(* CODESYS project mbc_Log4TC_tc3-4024_v0.2.1.library
   DefaultNamespace: log4tc
   DocFormat: reStructuredText
   Description: A library for logging in PLC code.
   Author: mbc engineering GmbH
   Title: log4TC
   Version: 0.2.1
   Company: mbc engineering GmbH
   Placeholder: log4TC

Project tree, tasks and I/O mapping:
  libraries: Base Interfaces, * (System); Tc2_Standard, * (Beckhoff Automation GmbH); Tc2_System, * (Beckhoff Automation GmbH); Tc2_Utilities, * (Beckhoff Automation GmbH); Tc3_Module, * (Beckhoff Automation GmbH); TcUnit, 1.0.0.0 (www.tcunit.org)
  API/
    Context/
      function F_LogContext [ST]
      function block FB_ScopedContext [ST]: Begin, ContextBuilder, End
      interface I_ContextBuilder: AddBool, AddByte, AddDInt, AddDWord, AddInt, AddLint, AddLReal, AddLWord, AddReal, AddSInt, AddString, AddUDInt, AddUInt, AddULint, AddUSInt, AddWord, Clear, Remove
    Full/
      function block FB_LoggerLAC [ST]: FB_init, LoggerContext
    Simple/
      Any/
        function F_LogA1 [ST]
        function F_LogA10 [ST]
        function F_LogA2 [ST]
        function F_LogA3 [ST]
        function F_LogA4 [ST]
        function F_LogA5 [ST]
        function F_LogA6 [ST]
        function F_LogA7 [ST]
        function F_LogA8 [ST]
        function F_LogA9 [ST]
        function F_LogLA1 [ST]
        function F_LogLA10 [ST]
        function F_LogLA10C [ST]
        function F_LogLA1C [ST]
        function F_LogLA2 [ST]
        function F_LogLA2C [ST]
        function F_LogLA3 [ST]
        function F_LogLA3C [ST]
        function F_LogLA4 [ST]
        function F_LogLA4C [ST]
        function F_LogLA5 [ST]
        function F_LogLA5C [ST]
        function F_LogLA6 [ST]
        function F_LogLA6C [ST]
        function F_LogLA7 [ST]
        function F_LogLA7C [ST]
        function F_LogLA8 [ST]
        function F_LogLA8C [ST]
        function F_LogLA9 [ST]
        function F_LogLA9C [ST]
      TArg/
        function F_LogL1 [ST]
        function F_LogL10 [ST]
        function F_LogL2 [ST]
        function F_LogL3 [ST]
        function F_LogL4 [ST]
        function F_LogL5 [ST]
        function F_LogL6 [ST]
        function F_LogL7 [ST]
        function F_LogL8 [ST]
        function F_LogL9 [ST]
      function F_Log [ST]
      function F_LogBuilder [ST]
      function F_LogC [ST]
      function F_LogL [ST]
      function F_LogLC [ST]
      interface I_LogBuilder: CreateLog, WithContextInt, WithIntArg, WithLogger, WithStringArg
    data type E_LogLevel
    program PRG_TaskLog [ST]: Call, Init, RtcTime, TaskContextBuilder, TaskLogger
  DUTs/
    data type E_CustomTypes
    data type E_Scope
    data type ST_Log4TcTaskInfo
    data type ST_ScopedContextStack
  GVLs/
    global variables Config
    global variables Const
    global variables Log4TcInfo
  ITFs/
    interface I_LogEntryAdder: AddToLogEntry
  POUs/
    Utils/
      function F_DINT_TO_UINT_MAX [ST]
      function block FB_LogBuffer [ST]: BufferFree, BufferPtr, BufferStartPtr, BufferUsed, Clear, DataAdded
      function block FB_RTC_Sync [ST]: Call, RtcTime
      function IncUDINT [ST]
    function F_InternalLog [ST]
    function F_LogA [ST]
    function F_LogTArg [ST]
    function block FB_ContextBuilder [ST]: _FindContext, _GetDataLen, _GetOffsetToData, _GetSize, _ReadName, _ReadType, AddBool, AddByte, AddDInt, AddDWord, AddInt, AddLInt, AddLReal, AddLWord, AddReal, AddSInt, AddString, AddUDInt, AddUInt, AddULInt, AddUSInt, AddWord, Clear, Remove, _BufferCount, _ContextCount, _GetContextOffset, _AddContext, _Copy, _RemoveContext, _ReplaceContext, _Reset, _WriteByte, _WriteInt, AddToLogEntry
    function block FB_Log4TcTask [ST]: _InitAndCheckTask, _ReadBuffer, Call, Init, TaskContext, WriteBuffer
    function block FB_LogEntry [ST]: _Copy, _Reset, _WriteByte, _WriteDInt, _WriteInt, _WriteLInt, _WriteString, _WriteUDInt, _WriteUInt, _WriteWString, AddAnyArg, AddBuffer, AddContext, AddTArg, End, Start
    program PRG_ScopedContextStack [ST]: TaskContextStack
  Test/
    function block FB_ContextBuilder_Test [ST]: AddInt_ShouldAddInt, AddInt_WithSameName_ShouldReplace, AddString_ShouldAddString, AddString_WithSameName_ShouldReAdd, AddString_WithSameName_ShouldReplace, RemoveInt_ShouldRemove, RemoveString_ShouldRemove
    program PRG_Test [ST]
  Version/
    global variables Global_Version
  program ApiTest [ST]
*)

// API/E_LogLevel
(*
:Description: Definition of available log levels. 

The log levels are ordered. ``eTrace`` has the lowest priority, ``eFatal`` has the
highest priority.

===============
Log Level Usage
===============

Is is recommended to build a guidline for consistent use of the log level. A example
could be the following:

:eFatal: The fatal level should be used for any error which will to malfunction of the most
	part of the program. Log message of this type must be handled immedialtely.
	
	Example: A Safety controller could not be initialised

:eError: The error level should be used when the program cannot continue to work properly.
	Normally this means that a operator/user has to be alerted and something has to
	be fixed.

	Example: Communication errors, something stops a process

:eWarn: The warn level should be used when some expected condition has happend, but the
	software can proceed in some way or the operation can be repeated later. Normaly
	the warn level should be read by the user/operator at some time, not necessarly 
	immediately.

	Example: Cannot connect to some external system (but will repeat to try)

:eInfo: The info level should track some of the import state changes in the programm. This
	information can be used by the user/operator on demand to track a problem.

	Example: A state of a state-machine has changed, a new recipe has been loaded

:eDebug: The info level should track of the some internals, normally only of importance to
	developers.

:eTrace: The trace level should be used to track some internal processing. This is rarely
	used, even by developers, mostly to track some difficult problem.

*)
{attribute 'qualified_only'}
{attribute 'strict'}
{attribute 'to_string'}
TYPE E_LogLevel :
(
	eTrace 	:= 0,	(* Trace log level. *)
	eDebug 	:= 1,	(* Debug log level. *)
	eInfo	:= 2,	(* Info log level. *)
	eWarn	:= 3,	(* Warn log level. *)
	eError	:= 4,	(* Error log level. *)
	eFatal	:= 5	(* Fatal log level. *)
) UINT;
END_TYPE

// DUTs/E_CustomTypes
{attribute 'qualified_only'}
{attribute 'strict'}
TYPE INTERNAL E_CustomTypes :
(
	eType_TIME				:= 20000,
	eType_LTIME				:= 20001,
	eType_DATE				:= 20002,
	eType_DATE_AND_TIME		:= 20003,
	eType_TIME_OF_DAY		:= 20004,
	eType_ENUM				:= 20005,
	eType_WSTRING			:= 20006
) INT;
END_TYPE

// DUTs/E_Scope

{attribute 'qualified_only'}
{attribute 'strict'}
{attribute 'conditionalshow'}
{attribute 'to_string'}
TYPE E_Scope :
(
	eLog			:= 0,
	eLogger			:= 1,
	eScoped			:= 2,
	eTask			:= 3
) BYTE;
END_TYPE

// DUTs/ST_Log4TcTaskInfo
TYPE ST_Log4TcTaskInfo :
STRUCT
	nAddLogToBuffer						: UDINT;	(* Counts number of logs added to message buffer. *)
	nAddLogToBufferErrorCount			: UDINT;	(* Counts error when adding log message to task buffer. *)
	nSendLogBufferErrorCount			: UDINT;	(* Counts error when sending log task buffer to service. *)
	nMaxUsedBufferSize					: UDINT;	(* Max. used buffer size of log task buffer. *)
END_STRUCT
END_TYPE

// DUTs/ST_ScopedContextStack
{attribute 'conditionalshow'}
TYPE INTERNAL ST_ScopedContextStack :
STRUCT
	aScopedContext		: ARRAY[0..Config.nMaxScopedContext-1] OF I_ContextBuilder;
	nScopeContextCount	: UINT (0..Config.nMaxScopedContext);
END_STRUCT
END_TYPE

// GVLs/Config
{attribute 'qualified_only'}
VAR_GLOBAL CONSTANT
	eInternalLog			: E_LogLevel := E_LogLevel.eInfo;	(* min. log level for internal logging. *)
	nBufferLen 				: UINT := 8192;		(* Length of per task log buffer in bytes *)
	nMaxScopedContext		: UINT := 4;		(* Max. number of nested scope context. *)
	sLicenseActivation		: STRING := '';	
END_VAR

// GVLs/Const
{attribute 'qualified_only'}
VAR_GLOBAL CONSTANT
	sGlobalLogger		: STRING := '_GLOBAL_';		(* Global logger name for logger without logger input *)
	sLoggerFromInstance	: STRING := '__INST__';		(* FB_Logger*: Initialize logger name from instance path. *)
END_VAR

// GVLs/Log4TcInfo
{attribute 'qualified_only'}
VAR_GLOBAL
	aTaskInfo							: ARRAY[1..SIZEOF(TwinCAT_SystemInfoVarList._TaskInfo)/SIZEOF(PlcTaskSystemInfo)] OF ST_Log4TcTaskInfo;
END_VAR

// Version/Global_Version
{attribute 'TcGenerated'}
{attribute 'no-analysis'}
{attribute 'linkalways'}
// This function has been automatically generated from the project information.
VAR_GLOBAL CONSTANT
	{attribute 'const_non_replaced'}
	stLibVersion_log4TC : ST_LibVersion := (iMajor := 0, iMinor := 2, iBuild := 1, iRevision := 0, nFlags := 0, sVersion := '0.2.1');
END_VAR

// API/Context/F_LogContext
FUNCTION F_LogContext : I_ContextBuilder
VAR_STAT
	aTaskContext		: ARRAY[1..SIZEOF(TwinCAT_SystemInfoVarList._TaskInfo)/SIZEOF(PlcTaskSystemInfo)] OF FB_ContextBuilder;
END_VAR

F_LogContext := aTaskContext[Tc2_System.GETCURTASKINDEXEX()].Clear();

END_FUNCTION

// API/Context/I_ContextBuilder
INTERFACE I_ContextBuilder EXTENDS __System.IQueryInterface

METHOD AddBool : I_ContextBuilder
VAR_INPUT
	sName		: T_MaxString;	
	bValue		: BOOL;
END_VAR
END_METHOD

METHOD AddByte : I_ContextBuilder
VAR_INPUT
	sName		: T_MaxString;
	nValue		: BYTE;
END_VAR
END_METHOD

METHOD AddDInt : I_ContextBuilder
VAR_INPUT
	sName		: T_MaxString;
	nValue		: DINT;
END_VAR
END_METHOD

METHOD AddDWord : I_ContextBuilder
VAR_INPUT
	sName	: Tc2_System.T_MaxString;
	nValue	: DWORD;
END_VAR
END_METHOD

METHOD AddInt : I_ContextBuilder
VAR_INPUT
	sName		: T_MaxString;
	nValue		: INT;
END_VAR
END_METHOD

METHOD AddLint : I_ContextBuilder
VAR_INPUT
	sName		: T_MaxString;
	nValue		: LINT;
END_VAR
END_METHOD

METHOD AddLReal : I_ContextBuilder
VAR_INPUT
	sName	: Tc2_System.T_MaxString;
	fValue	: LREAL;
END_VAR
END_METHOD

METHOD AddLWord : I_ContextBuilder
VAR_INPUT
	sName		: T_MaxString;
	nValue		: LWORD;
END_VAR
END_METHOD

METHOD AddReal : I_ContextBuilder
VAR_INPUT
	sName	: Tc2_System.T_MaxString;
	fValue	: REAL;
END_VAR
END_METHOD

METHOD AddSInt : I_ContextBuilder
VAR_INPUT
	sName		: T_MaxString;
	nValue		: SINT;
END_VAR
END_METHOD

METHOD AddString : I_ContextBuilder
VAR_INPUT
	sName		: T_MaxString;
	sValue		: T_MaxString;
END_VAR
END_METHOD

METHOD AddUDInt : I_ContextBuilder
VAR_INPUT
	sName		: T_MaxString;
	nValue		: UDINT;
END_VAR
END_METHOD

METHOD AddUInt : I_ContextBuilder
VAR_INPUT
	sName		: T_MaxString;
	nValue		: UINT;
END_VAR
END_METHOD

METHOD AddULint : I_ContextBuilder
VAR_INPUT
	sName		: T_MaxString;
	nValue		: ULINT;
END_VAR
END_METHOD

METHOD AddUSInt : I_ContextBuilder
VAR_INPUT
	sName		: T_MaxString;
	nValue		: USINT;
END_VAR
END_METHOD

METHOD AddWord : I_ContextBuilder
VAR_INPUT
	sName	: Tc2_System.T_MaxString;
	nValue	: WORD;
END_VAR
END_METHOD

METHOD Clear : I_ContextBuilder
VAR_INPUT
END_VAR
END_METHOD

METHOD Remove : I_ContextBuilder
VAR_INPUT
	sName	: Tc2_System.T_MaxString;
END_VAR
END_METHOD

END_INTERFACE

// POUs/FB_ContextBuilder
{attribute 'no_explicit_call' := 'no direct call necessary'}
{attribute 'conditionalshow'}
FUNCTION_BLOCK INTERNAL FB_ContextBuilder IMPLEMENTS I_ContextBuilder, I_LogEntryAdder
VAR CONSTANT
	nBufferSize			: UINT := 1024;
END_VAR
VAR
	aBuffer				: ARRAY[0..nBufferSize - 1] OF BYTE;	(* buffer for context variables *)
	nBufferCount		: UINT := 0;
	
	aContext			: ARRAY[0..19] OF UINT;
	nContextCount		: UINT(0..20) := 0;
END_VAR

METHOD PRIVATE _FindContext : UINT
VAR_INPUT
	refName		: REFERENCE TO Tc2_System.T_MaxString;
END_VAR
VAR
	nIdx		: UINT;
	nLen		: BYTE;
END_VAR
IF nContextCount > 0 THEN
	FOR nIdx := 0 TO nContextCount - 1 DO
		IF _ReadName(nIdx) = refName THEN
			_FindContext := nIdx;
			RETURN;
		END_IF
	END_FOR
END_IF

_FindContext := 16#FFFF;
END_METHOD

METHOD INTERNAL _GetDataLen : UINT
VAR_INPUT
	nIdx		: UINT;
END_VAR
VAR
	nSize		: UINT;
END_VAR
_GetDataLen := _GetSize(nIdx) - _GetOffsetToData(nIdx);
END_METHOD

METHOD PRIVATE _GetOffsetToData : UINT
VAR_INPUT
	nIdx		: UINT;
END_VAR
VAR
	pBuf		: PVOID;
	nOffset		: UINT;
END_VAR
pBuf := ADR(aBuffer) + aContext[nIdx];

// Offset to value (Skip name and type)
_GetOffsetToData := PBYTE_TO_BYTE(pBuf) + SIZEOF(BYTE) + SIZEOF(INT); // VARSTRING + INT
END_METHOD

METHOD PRIVATE _GetSize : UINT
VAR_INPUT
	nIdx		: UINT;
END_VAR
IF nIdx < nContextCount THEN
	IF (nIdx + 1) < nContextCount THEN
		_GetSize := aContext[nIdx + 1] - aContext[nIdx];
	ELSE
		_GetSize := nBufferCount - aContext[nIdx];
	END_IF
ELSE
	_GetSize := 0; 
END_IF
END_METHOD

METHOD INTERNAL _ReadName : T_MaxString
VAR_INPUT
	nIdx		: UINT;
END_VAR
VAR
	pBuf		: PVOID;
	nLen		: BYTE;
END_VAR
IF nIdx < nContextCount THEN
	pBuf := ADR(aBuffer) + aContext[nIdx];
	nLen := PBYTE_TO_BYTE(pBuf);
	MEMCPY(ADR(_ReadName), pBuf + 1, nLen);
	_ReadName[nLen] := 0;
ELSE
	_ReadName := '';	
END_IF
END_METHOD

METHOD INTERNAL _ReadType : INT
VAR_INPUT
	nIdx		: UINT;
END_VAR
VAR
	pBuf		: PVOID;
	nLen		: BYTE;
	nOffset		: UINT;
END_VAR
pBuf := ADR(aBuffer) + aContext[nIdx];

// Offset to value (Skip name and type)
nOffset := PBYTE_TO_BYTE(pBuf) + SIZEOF(BYTE); // VARSTRING + INT

MEMCPY(ADR(_ReadType), pBuf + nOffset, SIZEOF(INT));
END_METHOD

METHOD AddBool : I_ContextBuilder
VAR_INPUT
	sName		: T_MaxString;
	bValue		: BOOL;
END_VAR
VAR
	nIdx	: UINT;
END_VAR
AddBool := THIS^;

nIdx := _FindContext(sName);
IF nIdx <> 16#FFFF THEN
	IF _GetDataLen(nIdx) = SIZEOF(bValue) THEN
		_ReplaceContext(nIdx, Tc2_Utilities.E_ArgType.ARGTYPE_BOOL, ADR(bValue), SIZEOF(bValue));
		RETURN;
	END_IF
	
	_RemoveContext(sName);
END_IF

_AddContext(
	refName		:= sName,
	nValueType	:= Tc2_Utilities.E_ArgType.ARGTYPE_BOOL,
	pValue		:= ADR(bValue),
	nValueLen	:= SIZEOF(bValue)
);
END_METHOD

METHOD AddByte : I_ContextBuilder
VAR_INPUT
	sName		: T_MaxString;
	nValue		: BYTE;
END_VAR
VAR
	nIdx	: UINT;
END_VAR
AddByte := THIS^;

nIdx := _FindContext(sName);
IF nIdx <> 16#FFFF THEN
	IF _GetDataLen(nIdx) = SIZEOF(nValue) THEN
		_ReplaceContext(nIdx, Tc2_Utilities.E_ArgType.ARGTYPE_BYTE, ADR(nValue), SIZEOF(nValue));
		RETURN;
	END_IF
	
	_RemoveContext(sName);
END_IF

_AddContext(
	refName		:= sName,
	nValueType	:= Tc2_Utilities.E_ArgType.ARGTYPE_BYTE,
	pValue		:= ADR(nValue),
	nValueLen	:= SIZEOF(nValue)
);
END_METHOD

METHOD AddDInt : I_ContextBuilder
VAR_INPUT
	sName	: Tc2_System.T_MaxString;
	nValue	: DINT;
END_VAR
VAR
	nIdx	: UINT;
END_VAR
AddDInt := THIS^;

nIdx := _FindContext(sName);
IF nIdx <> UINT#16#FFFF THEN
	IF _GetDataLen(nIdx) = SIZEOF(nValue) THEN
		_ReplaceContext(nIdx, Tc2_Utilities.E_ArgType.ARGTYPE_DINT, ADR(nValue), SIZEOF(nValue));
		RETURN;
	END_IF
	
	_RemoveContext(sName);
END_IF

_AddContext(
	refName		:= sName,
	nValueType	:= Tc2_Utilities.E_ArgType.ARGTYPE_DINT,
	pValue		:= ADR(nValue),
	nValueLen	:= SIZEOF(nValue)
);
END_METHOD

METHOD AddDWord : I_ContextBuilder
VAR_INPUT
	sName	: Tc2_System.T_MaxString;
	nValue	: DWORD;
END_VAR
VAR
	nIdx	: UINT;
END_VAR
AddDWord := THIS^;

nIdx := _FindContext(sName);
IF nIdx <> 16#FFFF THEN
	IF _GetDataLen(nIdx) = SIZEOF(nValue) THEN
		_ReplaceContext(nIdx, Tc2_Utilities.E_ArgType.ARGTYPE_DWORD, ADR(nValue), SIZEOF(nValue));
		RETURN;
	END_IF
	
	_RemoveContext(sName);
END_IF

_AddContext(
	refName		:= sName,
	nValueType	:= Tc2_Utilities.E_ArgType.ARGTYPE_DWORD,
	pValue		:= ADR(nValue),
	nValueLen	:= SIZEOF(nValue)
);
END_METHOD

METHOD AddInt : I_ContextBuilder
VAR_INPUT
	sName	: Tc2_System.T_MaxString;
	nValue	: INT;
END_VAR
VAR
	nIdx	: UINT;
END_VAR
AddInt := THIS^;

nIdx := _FindContext(sName);
IF nIdx <> UINT#16#FFFF THEN
	IF _GetDataLen(nIdx) = SIZEOF(nValue) THEN
		_ReplaceContext(nIdx, Tc2_Utilities.E_ArgType.ARGTYPE_INT, ADR(nValue), SIZEOF(nValue));
		RETURN;
	END_IF
	
	_RemoveContext(sName);
END_IF

_AddContext(
	refName		:= sName,
	nValueType	:= Tc2_Utilities.E_ArgType.ARGTYPE_INT,
	pValue		:= ADR(nValue),
	nValueLen	:= SIZEOF(nValue)
);
END_METHOD

METHOD AddLInt : I_ContextBuilder
VAR_INPUT
	sName	: Tc2_System.T_MaxString;
	nValue	: LINT;
END_VAR
VAR
	nIdx	: UINT;
END_VAR
AddLInt := THIS^;

nIdx := _FindContext(sName);
IF nIdx <> UINT#16#FFFF THEN
	IF _GetDataLen(nIdx) = SIZEOF(nValue) THEN
		_ReplaceContext(nIdx, Tc2_Utilities.E_ArgType.ARGTYPE_LARGE, ADR(nValue), SIZEOF(nValue));
		RETURN;
	END_IF
	
	_RemoveContext(sName);
END_IF

_AddContext(
	refName		:= sName,
	nValueType	:= Tc2_Utilities.E_ArgType.ARGTYPE_LARGE,
	pValue		:= ADR(nValue),
	nValueLen	:= SIZEOF(nValue)
);
END_METHOD

METHOD AddLReal : I_ContextBuilder
VAR_INPUT
	sName	: Tc2_System.T_MaxString;
	fValue	: LREAL;
END_VAR
VAR
	nIdx	: UINT;
END_VAR
AddLReal := THIS^;

nIdx := _FindContext(sName);
IF nIdx <> 16#FFFF THEN
	IF _GetDataLen(nIdx) = SIZEOF(fValue) THEN
		_ReplaceContext(nIdx, Tc2_Utilities.E_ArgType.ARGTYPE_LREAL, ADR(fValue), SIZEOF(fValue));
		RETURN;
	END_IF
	
	_RemoveContext(sName);
END_IF

_AddContext(
	refName		:= sName,
	nValueType	:= Tc2_Utilities.E_ArgType.ARGTYPE_LREAL,
	pValue		:= ADR(fValue),
	nValueLen	:= SIZEOF(fValue)
);
END_METHOD

METHOD AddLWord : I_ContextBuilder
VAR_INPUT
	sName	: Tc2_System.T_MaxString;
	nValue	: LWORD;
END_VAR
VAR
	nIdx	: UINT;
END_VAR
AddLWord := THIS^;

nIdx := _FindContext(sName);
IF nIdx <> UINT#16#FFFF THEN
	IF _GetDataLen(nIdx) = SIZEOF(nValue) THEN
		_ReplaceContext(nIdx, Tc2_Utilities.E_ArgType.ARGTYPE_LWORD, ADR(nValue), SIZEOF(nValue));
		RETURN;
	END_IF
	
	_RemoveContext(sName);
END_IF

_AddContext(
	refName		:= sName,
	nValueType	:= Tc2_Utilities.E_ArgType.ARGTYPE_LWORD,
	pValue		:= ADR(nValue),
	nValueLen	:= SIZEOF(nValue)
);
END_METHOD

METHOD AddReal : I_ContextBuilder
VAR_INPUT
	sName	: Tc2_System.T_MaxString;
	fValue	: REAL;
END_VAR
VAR
	nIdx	: UINT;
END_VAR
AddReal := THIS^;

nIdx := _FindContext(sName);
IF nIdx <> 16#FFFF THEN
	IF _GetDataLen(nIdx) = SIZEOF(fValue) THEN
		_ReplaceContext(nIdx, Tc2_Utilities.E_ArgType.ARGTYPE_REAL, ADR(fValue), SIZEOF(fValue));
		RETURN;
	END_IF
	
	_RemoveContext(sName);
END_IF

_AddContext(
	refName		:= sName,
	nValueType	:= Tc2_Utilities.E_ArgType.ARGTYPE_REAL,
	pValue		:= ADR(fValue),
	nValueLen	:= SIZEOF(fValue)
);
END_METHOD

METHOD AddSInt : I_ContextBuilder
VAR_INPUT
	sName	: Tc2_System.T_MaxString;
	nValue	: SINT;
END_VAR
VAR
	nIdx	: UINT;
END_VAR
AddSInt := THIS^;

nIdx := _FindContext(sName);
IF nIdx <> UINT#16#FFFF THEN
	IF _GetDataLen(nIdx) = SIZEOF(nValue) THEN
		_ReplaceContext(nIdx, Tc2_Utilities.E_ArgType.ARGTYPE_SINT, ADR(nValue), SIZEOF(nValue));
		RETURN;
	END_IF
	
	_RemoveContext(sName);
END_IF

_AddContext(
	refName		:= sName,
	nValueType	:= Tc2_Utilities.E_ArgType.ARGTYPE_SINT,
	pValue		:= ADR(nValue),
	nValueLen	:= SIZEOF(nValue)
);
END_METHOD

METHOD AddString : I_ContextBuilder
VAR_INPUT
	sName		: T_MaxString;
	sValue		: T_MaxString;
END_VAR
VAR
	nIdx		: UINT;
	aDataBuffer	: ARRAY[0..255] OF BYTE;
	nLen		: INT;
END_VAR
AddString := THIS^;

nLen := LEN(sValue);
IF nLen >= 0 AND nLen <= 255 THEN
	// copy string with length-byte into temporary buffer
	aDataBuffer[0] := INT_TO_BYTE(nLen);
	MEMCPY(ADR(aDataBuffer) + 1, ADR(sValue), INT_TO_UDINT(nLen));
	
	nIdx := _FindContext(sName);
	IF nIdx <> UINT#16#FFFF THEN
		IF _GetDataLen(nIdx) = INT_TO_UINT(nLen + 1) THEN
			_ReplaceContext(nIdx, Tc2_Utilities.E_ArgType.ARGTYPE_STRING, ADR(aDataBuffer), INT_TO_UINT(nLen) + 1);
			RETURN;
		END_IF
		
		_RemoveContext(sName);
	END_IF
	
	_AddContext(
		refName		:= sName,
		nValueType	:= E_ArgType.ARGTYPE_STRING,
		pValue		:= ADR(aDataBuffer),
		nValueLen	:= INT_TO_UINT(nLen) + 1
	);
ELSE
	F_InternalLog(
		E_LogLEvel.eFatal,
		'FB_ContextBuilder.AddString',
		'Pre check failed - string is longer than 255 (%d)',
		Tc2_Utilities.F_INT(nLen),
		Tc2_Utilities.EMPTY_ARG_VALUE,
		Tc2_Utilities.EMPTY_ARG_VALUE,
		Tc2_Utilities.EMPTY_ARG_VALUE
	);
END_IF
END_METHOD

METHOD AddUDInt : I_ContextBuilder
VAR_INPUT
	sName	: Tc2_System.T_MaxString;
	nValue	: UDINT;
END_VAR
VAR
	nIdx	: UINT;
END_VAR
AddUDInt := THIS^;

nIdx := _FindContext(sName);
IF nIdx <> UINT#16#FFFF THEN
	IF _GetDataLen(nIdx) = SIZEOF(nValue) THEN
		_ReplaceContext(nIdx, Tc2_Utilities.E_ArgType.ARGTYPE_UDINT, ADR(nValue), SIZEOF(nValue));
		RETURN;
	END_IF
	
	_RemoveContext(sName);
END_IF

_AddContext(
	refName		:= sName,
	nValueType	:= Tc2_Utilities.E_ArgType.ARGTYPE_UDINT,
	pValue		:= ADR(nValue),
	nValueLen	:= SIZEOF(nValue)
);
END_METHOD

METHOD AddUInt : I_ContextBuilder
VAR_INPUT
	sName	: Tc2_System.T_MaxString;
	nValue	: UINT;
END_VAR
VAR
	nIdx	: UINT;
END_VAR
AddUInt := THIS^;

nIdx := _FindContext(sName);
IF nIdx <> UINT#16#FFFF THEN
	IF _GetDataLen(nIdx) = SIZEOF(nValue) THEN
		_ReplaceContext(nIdx, Tc2_Utilities.E_ArgType.ARGTYPE_UINT, ADR(nValue), SIZEOF(nValue));
		RETURN;
	END_IF
	
	_RemoveContext(sName);
END_IF

_AddContext(
	refName		:= sName,
	nValueType	:= Tc2_Utilities.E_ArgType.ARGTYPE_UINT,
	pValue		:= ADR(nValue),
	nValueLen	:= SIZEOF(nValue)
);
END_METHOD

METHOD AddULInt : I_ContextBuilder
VAR_INPUT
	sName	: Tc2_System.T_MaxString;
	nValue	: ULINT;
END_VAR
VAR
	nIdx	: UINT;
END_VAR
AddULInt := THIS^;

nIdx := _FindContext(sName);
IF nIdx <> UINT#16#FFFF THEN
	IF _GetDataLen(nIdx) = SIZEOF(nValue) THEN
		_ReplaceContext(nIdx, Tc2_Utilities.E_ArgType.ARGTYPE_ULARGE, ADR(nValue), SIZEOF(nValue));
		RETURN;
	END_IF
	
	_RemoveContext(sName);
END_IF

_AddContext(
	refName		:= sName,
	nValueType	:= Tc2_Utilities.E_ArgType.ARGTYPE_ULARGE,
	pValue		:= ADR(nValue),
	nValueLen	:= SIZEOF(nValue)
);
END_METHOD

METHOD AddUSInt : I_ContextBuilder
VAR_INPUT
	sName	: Tc2_System.T_MaxString;
	nValue	: USINT;
END_VAR
VAR
	nIdx	: UINT;
END_VAR
AddUSInt := THIS^;

nIdx := _FindContext(sName);
IF nIdx <> UINT#16#FFFF THEN
	IF _GetDataLen(nIdx) = SIZEOF(nValue) THEN
		_ReplaceContext(nIdx, Tc2_Utilities.E_ArgType.ARGTYPE_USINT, ADR(nValue), SIZEOF(nValue));
		RETURN;
	END_IF
	
	_RemoveContext(sName);
END_IF

_AddContext(
	refName		:= sName,
	nValueType	:= Tc2_Utilities.E_ArgType.ARGTYPE_USINT,
	pValue		:= ADR(nValue),
	nValueLen	:= SIZEOF(nValue)
);
END_METHOD

METHOD AddWord : I_ContextBuilder
VAR_INPUT
	sName	: Tc2_System.T_MaxString;
	nValue	: WORD;
END_VAR
VAR
	nIdx	: UINT;
END_VAR
AddWord := THIS^;

nIdx := _FindContext(sName);
IF nIdx <> 16#FFFF THEN
	IF _GetDataLen(nIdx) = SIZEOF(nValue) THEN
		_ReplaceContext(nIdx, Tc2_Utilities.E_ArgType.ARGTYPE_WORD, ADR(nValue), SIZEOF(nValue));
		RETURN;
	END_IF
	
	_RemoveContext(sName);
END_IF

_AddContext(
	refName		:= sName,
	nValueType	:= Tc2_Utilities.E_ArgType.ARGTYPE_WORD,
	pValue		:= ADR(nValue),
	nValueLen	:= SIZEOF(nValue)
);
END_METHOD

METHOD Clear : I_ContextBuilder
VAR_INPUT
END_VAR
_Reset();
Clear := THIS^;
END_METHOD

METHOD Remove : I_ContextBuilder
VAR_INPUT
	sName	: Tc2_System.T_MaxString;
END_VAR
Remove := THIS^;
_RemoveContext(sName);
END_METHOD

PROPERTY INTERNAL _BufferCount : UINT
GET
_BufferCount := nBufferCount;
END_GET
END_PROPERTY

PROPERTY INTERNAL _ContextCount : UINT
GET
_ContextCount := nContextCount;
END_GET
END_PROPERTY

METHOD INTERNAL _GetContextOffset : UINT
VAR_INPUT
	nIdx		: UINT;
END_VAR
_GetContextOffset := aContext[nIdx];
END_METHOD

METHOD PRIVATE _AddContext : BOOL
VAR_INPUT
	refName			: REFERENCE TO T_MaxString;
	nValueType		: INT;
	pValue			: PVOID;
	nValueLen		: UINT;
END_VAR
VAR
	nContextSize	: UINT;
	nNameLen		: INT;
	bOk				: BOOL;
END_VAR
_AddContext := FALSE;

IF nContextCount < 20 THEN
	nNameLen := Tc2_Standard.LEN(refName);
	IF nNameLen >= 0 AND nNameLen <= 255 THEN
		nContextSize :=
			INT_TO_UINT(nNameLen + 1) 		// String + Length-Byte
			+ INT_TO_UINT(SIZEOF(INT))		// Value type
			+ nValueLen;		// Value length

		IF (nBufferSize - nBufferCount) >= nContextSize  THEN
			aContext[nContextCount] := nBufferCount;
			nContextCount := nContextCount + 1;
		
			bOk :=
				_WriteByte(INT_TO_BYTE(nNameLen)) AND_THEN 
				_Copy(ADR(refName), INT_TO_UINT(nNameLen)) AND_THEN
				_WriteInt(nValueType) AND_THEN
				_Copy(pValue, nValueLen);
			
			IF bOk THEN
				_AddContext := TRUE;
			ELSE
				// Rollback
				nContextCount := nContextCount - 1;
				nBufferCount := aContext[nContextCount];
				
				F_InternalLog(
					E_LogLevel.eFatal,
					'FB_ContextBuilder._AddContext',
					'Error copy data to buffer - should not happen because of precheck',
					Tc2_Utilities.EMPTY_ARG_VALUE,
					Tc2_Utilities.EMPTY_ARG_VALUE,
					Tc2_Utilities.EMPTY_ARG_VALUE,
					Tc2_Utilities.EMPTY_ARG_VALUE
				);				
			END_IF
		ELSE
			F_InternalLog(
				E_LogLevel.eWarn,
				'FB_ContextBuilder._AddContext',
				'Too less space for adding context value %s.',
				Tc2_Utilities.F_StringEx(refName),
				Tc2_Utilities.EMPTY_ARG_VALUE,
				Tc2_Utilities.EMPTY_ARG_VALUE,
				Tc2_Utilities.EMPTY_ARG_VALUE
			);					
		END_IF
	ELSE
		// should not happen because T_MaxString is <= 255 bytes long
		F_InternalLog(
			E_LogLevel.eError,
			'FB_ContextBuilder._AddContext',
			'String longer than 255 bytes (actual=%d) - missin 0-byte?',
			Tc2_Utilities.F_INT(nNameLen),
			Tc2_Utilities.EMPTY_ARG_VALUE,
			Tc2_Utilities.EMPTY_ARG_VALUE,
			Tc2_Utilities.EMPTY_ARG_VALUE
		);		
	END_IF
ELSE
	F_InternalLog(
		E_LogLevel.eWarn,
		'FB_ContextBuilder._AddContext',
		'Number of context variable exceed (max. 20).',
		Tc2_Utilities.EMPTY_ARG_VALUE,
		Tc2_Utilities.EMPTY_ARG_VALUE,
		Tc2_Utilities.EMPTY_ARG_VALUE,
		Tc2_Utilities.EMPTY_ARG_VALUE
	);		
END_IF
END_METHOD

METHOD PRIVATE _Copy : BOOL
VAR_INPUT
	pSrc		: PVOID;
	nCount		: UINT;
END_VAR
IF (nBufferSize - nBufferCount) >= nCount THEN
	MEMCPY(ADR(aBuffer) + nBufferCount, pSrc, nCount);
	nBufferCount := nBufferCount + nCount;
	
	_Copy := TRUE;
ELSE
	_Copy := FALSE;
END_IF
END_METHOD

METHOD PRIVATE _RemoveContext : BOOL
VAR_INPUT
	refName		: REFERENCE TO Tc2_System.T_MaxString;
END_VAR
VAR
	nIdx		: UINT;
	nBufferOff	: UINT;
END_VAR
IF nContextCount > 0 THEN
	nIdx := _FindContext(refName);
	IF nIdx <> UINT#16#FFFF THEN
		(* Found - remove entry and compact buffer *)
		IF (nIdx + 1) < nContextCount THEN
			// Move buffer data
			MEMMOVE(
				ADR(aBuffer) + aContext[nIdx], 
				ADR(aBuffer) + aContext[nIdx + 1], 
				nBufferCount - aContext[nIdx + 1]
			);
			
			nBufferOff := aContext[nIdx + 1] - aContext[nIdx];
			nBufferCount := nBufferCount - nBufferOff;
			
			// Move and change index
			WHILE (nIdx + 1) < nContextCount DO
				aContext[nIdx] := aContext[nIdx + 1] - nBufferOff;
				nIdx := nIdx + 1;
			END_WHILE
		END_IF

		nContextCount := nContextCount - 1;
		_RemoveContext := TRUE;
		RETURN;
	END_IF
END_IF

_RemoveContext := FALSE;
END_METHOD

METHOD PRIVATE _ReplaceContext : BOOL
VAR_INPUT
	nIdx			: UINT;
	nValueType		: INT;
	pValue			: PVOID;
	nValueLen		: UINT;
END_VAR
VAR
	pBuf			: PVOID;
	nNameLen		: BYTE;
END_VAR
pBuf := ADR(aBuffer) + aContext[nIdx];

// Skip Name
nNameLen := PBYTE_TO_BYTE(pBuf);
pBuf := pBuf + nNameLen + 1;

pBuf := pBuf + MEMCPY(pBuf, ADR(nValueType), SIZEOF(nValueType));
pBuf := pBuf + MEMCPY(pBuf, pValue, nValueLen);
END_METHOD

METHOD PRIVATE _Reset
VAR_INPUT
END_VAR
nBufferCount := 0;
nContextCount := 0;
END_METHOD

METHOD PRIVATE _WriteByte : BOOL
VAR_INPUT
	nValue		: BYTE;
END_VAR
_WriteByte := _Copy(ADR(nValue), SIZEOF(nValue));
END_METHOD

METHOD PRIVATE _WriteInt : BOOL
VAR_INPUT
	nValue		: INT;
END_VAR
_WriteInt := _Copy(ADR(nValue), SIZEOF(nValue));
END_METHOD

METHOD AddToLogEntry : BOOL
VAR_INPUT
	eScope			: E_Scope;
	refLogEntry		: REFERENCE TO FB_LogEntry;
END_VAR
VAR
	nIdx			: UINT;
	bOk				: BOOL;
	nContextLen		: UINT;
END_VAR
nIdx := 0;
bOk := TRUE;
WHILE nIdx < nContextCount AND bOk DO
	refLogEntry.AddContext(eScope, ADR(aBuffer) + aContext[nIdx], _GetSize(nIdx));
	nIdx := nIdx + 1;
END_WHILE

IF nIdx < nContextCount AND NOT bOk THEN
	F_InternalLog(
		E_LogLevel.eWarn,
		'FB_ContextBuilder.AddLogEntry',
		'Could not add all context properties to log entry. (act=%d, all=%d)',
		Tc2_Utilities.F_UINT(nIdx),
		Tc2_Utilities.F_UINT(nContextCount),
		Tc2_Utilities.EMPTY_ARG_VALUE,
		Tc2_Utilities.EMPTY_ARG_VALUE
	);
END_IF 

AddToLogEntry := bOk;
END_METHOD

END_FUNCTION_BLOCK

// ITFs/I_LogEntryAdder
{attribute 'conditionalshow'}
INTERFACE INTERNAL I_LogEntryAdder EXTENDS __System.IQueryInterface

METHOD AddToLogEntry : BOOL
VAR_INPUT
	eScope			: E_Scope;
	refLogEntry		: REFERENCE TO FB_LogEntry;
END_VAR
END_METHOD

END_INTERFACE

// POUs/FB_LogEntry
{attribute 'no_explicit_call' := 'no direct call necessary'} 
{attribute 'conditionalshow'}
FUNCTION_BLOCK INTERNAL FB_LogEntry
VAR
	pBuffer				: PVOID;	// pointer to the current message buffer
	nBufferCount		: UINT;		// number of bytes written to the message buffer
	nBufferRemaining	: UINT;		// remaining bytes in the message buffer
	bError				: BOOL;		// indicates an error in the current message building
END_VAR

METHOD PRIVATE _Copy
VAR_INPUT
	pSrc		: PVOID;
	nCount		: UINT;
END_VAR
IF NOT bError AND_THEN nBufferRemaining >= nCount THEN
	Tc2_System.MEMCPY(pBuffer + nBufferCount, pSrc, nCount);
	nBufferCount := nBufferCount + nCount;
	nBufferRemaining := nBufferRemaining - nCount;
ELSE
	IF NOT bError THEN
		F_InternalLog(
			E_LogLevel.eWarn,
			'FB_LogEntry._Copy',
			'Error buffer overflow for log message (act=%d, new=%d)',
			Tc2_Utilities.F_UINT(nBufferCount),
			Tc2_Utilities.F_UINT(nCount),
			Tc2_Utilities.EMPTY_ARG_VALUE,
			Tc2_Utilities.EMPTY_ARG_VALUE
		);
	END_IF
	bError := TRUE;
END_IF
END_METHOD

METHOD PRIVATE _Reset
VAR
	pWriteBuffer	: POINTER TO FB_LogBuffer;
END_VAR
pWriteBuffer := PRG_TaskLog.TaskLogger.WriteBuffer;
pBuffer := pWriteBuffer^.BufferPtr;
nBufferCount := 0;
nBufferRemaining := pWriteBuffer^.BufferFree;

bError := FALSE;
END_METHOD

METHOD PRIVATE _WriteByte 
VAR_INPUT
	nValue		: BYTE;
END_VAR
_Copy(ADR(nValue), SIZEOF(nValue));
END_METHOD

METHOD PRIVATE _WriteDInt
VAR_INPUT
	nValue		: DINT;
END_VAR
_Copy(ADR(nValue), SIZEOF(nValue));
END_METHOD

METHOD PRIVATE _WriteInt 
VAR_INPUT
	nValue		: INT;
END_VAR
_Copy(ADR(nValue), SIZEOF(nValue));
END_METHOD

METHOD PRIVATE _WriteLInt
VAR_INPUT
	nValue		: LINT;
END_VAR
_Copy(ADR(nValue), SIZEOF(nValue));
END_METHOD

METHOD PRIVATE _WriteString
VAR_INPUT
	pValue		: POINTER TO Tc2_Utilities.T_MaxString;
END_VAR
VAR
	nLen			: INT;
END_VAR
IF pValue <> 0 THEN
	nLen := Tc2_Standard.LEN(pValue^);
	IF nLen >= 0 AND nLen <= 255 THEN
		_WriteByte(INT_TO_BYTE(nLen)); 
		_Copy(pValue, INT_TO_UINT(nLen));
	ELSE
		// should not happen because T_MaxString is <= 255 bytes long
		bError := TRUE;
		F_InternalLog(
			E_LogLevel.eError,
			'FB_LogEntry._WriteString',
			'String longer than 255 bytes (actual=%d) - missin 0-byte?',
			Tc2_Utilities.F_INT(nLen),
			Tc2_Utilities.EMPTY_ARG_VALUE,
			Tc2_Utilities.EMPTY_ARG_VALUE,
			Tc2_Utilities.EMPTY_ARG_VALUE
		);
	END_IF
ELSE
		bError := TRUE;
		F_InternalLog(
			E_LogLevel.eError,
			'FB_LogEntry._WriteString',
			'String null pointer',
			Tc2_Utilities.EMPTY_ARG_VALUE,
			Tc2_Utilities.EMPTY_ARG_VALUE,
			Tc2_Utilities.EMPTY_ARG_VALUE,
			Tc2_Utilities.EMPTY_ARG_VALUE
		);
END_IF
END_METHOD

METHOD PRIVATE _WriteUDInt
VAR_INPUT
	nValue		: UDINT;
END_VAR
_Copy(ADR(nValue), SIZEOF(nValue));
END_METHOD

METHOD PRIVATE _WriteUInt 
VAR_INPUT
	nValue		: UINT;
END_VAR
_Copy(ADR(nValue), SIZEOF(nValue));
END_METHOD

METHOD PRIVATE _WriteWString
VAR_INPUT
	pValue		: POINTER TO WSTRING(255);
END_VAR
VAR
	nLen			: INT;
END_VAR
IF pValue <> 0 THEN
	nLen := Tc2_Standard.WLEN(pValue^);
	IF nLen >= 0 AND nLen <= 255 THEN
		_WriteByte(INT_TO_BYTE(nLen)); 
		_Copy(pValue, INT_TO_UINT(nLen) * 2);
	ELSE
		// should not happen because T_MaxString is <= 255 bytes long
		bError := TRUE;
		F_InternalLog(
			E_LogLevel.eError,
			'FB_LogEntry._WriteWString',
			'String longer than 255 bytes (actual=%d) - missin 0-byte?',
			Tc2_Utilities.F_INT(nLen),
			Tc2_Utilities.EMPTY_ARG_VALUE,
			Tc2_Utilities.EMPTY_ARG_VALUE,
			Tc2_Utilities.EMPTY_ARG_VALUE
		);
	END_IF
ELSE
		bError := TRUE;
		F_InternalLog(
			E_LogLevel.eError,
			'FB_LogEntry._WriteWString',
			'String null pointer',
			Tc2_Utilities.EMPTY_ARG_VALUE,
			Tc2_Utilities.EMPTY_ARG_VALUE,
			Tc2_Utilities.EMPTY_ARG_VALUE,
			Tc2_Utilities.EMPTY_ARG_VALUE
		);
END_IF
END_METHOD

METHOD INTERNAL AddAnyArg : BOOL
VAR_INPUT
	nArgNo		: BYTE;
	stArg		: ANY;
END_VAR
VAR
	nLen		: INT;
END_VAR
IF bError THEN
	RETURN;
END_IF

IF stArg.pValue = 0 THEN
	RETURN;
END_IF

_WriteByte(1); // Type 1: Argument follows
_WriteByte(nArgno);

CASE stArg.TypeClass OF
	__SYSTEM.TYPE_CLASS.TYPE_BOOL:
		_WriteInt(Tc2_Utilities.E_ArgType.ARGTYPE_BOOL);
		IF Tc2_Utilities.PBYTE_TO_BYTE(stArg.pValue) <> 0 THEN
			_WriteByte(1);
		ELSE
			_WriteByte(0);
		END_IF

	__SYSTEM.TYPE_CLASS.TYPE_BYTE:
		_WriteInt(Tc2_Utilities.E_ArgType.ARGTYPE_BYTE);
		_Copy(stArg.pValue, SIZEOF(BYTE));
	
	__SYSTEM.TYPE_CLASS.TYPE_WORD:
		_WriteInt(Tc2_Utilities.E_ArgType.ARGTYPE_WORD);
		_Copy(stArg.pValue, SIZEOF(WORD));		
	
	__SYSTEM.TYPE_CLASS.TYPE_DWORD:
		_WriteInt(Tc2_Utilities.E_ArgType.ARGTYPE_DWORD);
		_Copy(stArg.pValue, SIZEOF(DWORD));		
	
	__SYSTEM.TYPE_CLASS.TYPE_LWORD:
		_WriteInt(Tc2_Utilities.E_ArgType.ARGTYPE_LWORD);
		_Copy(stArg.pValue, SIZEOF(LWORD));
	
	__SYSTEM.TYPE_CLASS.TYPE_SINT:
		_WriteInt(Tc2_Utilities.E_ArgType.ARGTYPE_SINT);
		_Copy(stArg.pValue, SIZEOF(SINT));
	
	__SYSTEM.TYPE_CLASS.TYPE_INT:
		_WriteInt(Tc2_Utilities.E_ArgType.ARGTYPE_INT);
		_Copy(stArg.pValue, SIZEOF(INT));		
	
	__SYSTEM.TYPE_CLASS.TYPE_DINT:
		_WriteInt(Tc2_Utilities.E_ArgType.ARGTYPE_DINT);
		_Copy(stArg.pValue, SIZEOF(DINT));		
	
	__SYSTEM.TYPE_CLASS.TYPE_LINT:
		_WriteInt(Tc2_Utilities.E_ArgType.ARGTYPE_LARGE);
		_Copy(stArg.pValue, SIZEOF(LINT));		
	
	__SYSTEM.TYPE_CLASS.TYPE_USINT:
		_WriteInt(Tc2_Utilities.E_ArgType.ARGTYPE_USINT);
		_Copy(stArg.pValue, SIZEOF(USINT));
	
	__SYSTEM.TYPE_CLASS.TYPE_UINT:
		_WriteInt(Tc2_Utilities.E_ArgType.ARGTYPE_UINT);
		_Copy(stArg.pValue, SIZEOF(UINT));		
	
	__SYSTEM.TYPE_CLASS.TYPE_UDINT:
		_WriteInt(Tc2_Utilities.E_ArgType.ARGTYPE_UDINT);
		_Copy(stArg.pValue, SIZEOF(UDINT));		
	
	__SYSTEM.TYPE_CLASS.TYPE_ULINT:
		_WriteInt(Tc2_Utilities.E_ArgType.ARGTYPE_ULARGE);
		_Copy(stArg.pValue, SIZEOF(ULINT));		
	
	__SYSTEM.TYPE_CLASS.TYPE_REAL:
		_WriteInt(Tc2_Utilities.E_ArgType.ARGTYPE_REAL);
		_Copy(stArg.pValue, SIZEOF(REAL));		
	
	__SYSTEM.TYPE_CLASS.TYPE_LREAL:
		_WriteInt(Tc2_Utilities.E_ArgType.ARGTYPE_LREAL);
		_Copy(stArg.pValue, SIZEOF(LREAL));		
	
	__SYSTEM.TYPE_CLASS.TYPE_STRING:
		_WriteInt(Tc2_Utilities.E_ArgType.ARGTYPE_STRING);
		_WriteString(stArg.pValue);

	__SYSTEM.TYPE_CLASS.TYPE_WSTRING:
		_WriteInt(E_CustomTypes.eType_WSTRING);
		_WriteWString(stArg.pValue);

	__SYSTEM.TYPE_CLASS.TYPE_TIME:
		_WriteInt(E_CustomTypes.eType_TIME);
		_Copy(stArg.pValue, SIZEOF(TIME));	

	__SYSTEM.TYPE_CLASS.TYPE_DATE:
		_WriteInt(E_CustomTypes.eType_DATE);
		_Copy(stArg.pValue, SIZEOF(DATE));		

	__SYSTEM.TYPE_CLASS.TYPE_DATEANDTIME:
		_WriteInt(E_CustomTypes.eType_DATE_AND_TIME);
		_Copy(stArg.pValue, SIZEOF(DATE_AND_TIME));		

	__SYSTEM.TYPE_CLASS.TYPE_TIMEOFDAY:
		_WriteInt(E_CustomTypes.eType_TIME_OF_DAY);
		_Copy(stArg.pValue, SIZEOF(TIME_OF_DAY));		

	__SYSTEM.TYPE_CLASS.TYPE_ENUM:
		_WriteInt(E_CustomTypes.eType_ENUM);
		// First write the integer value of the enumeration, expected 1 to 8 bytes
		CASE stArg.diSize OF
			1: 
				_WriteInt(Tc2_Utilities.E_ArgType.ARGTYPE_BYTE);
				_Copy(stArg.pValue, SIZEOF(BYTE));
			2:
				_WriteInt(Tc2_Utilities.E_ArgType.ARGTYPE_WORD);
				_Copy(stArg.pValue, SIZEOF(WORD));
			4:
				_WriteInt(Tc2_Utilities.E_ArgType.ARGTYPE_DWORD);
				_Copy(stArg.pValue, SIZEOF(DWORD));
			5:
				_WriteInt(Tc2_Utilities.E_ArgType.ARGTYPE_LWORD);
				_Copy(stArg.pValue, SIZEOF(LWORD));
			ELSE
				_WriteInt(Tc2_Utilities.E_ArgType.ARGTYPE_UNKNOWN);
		END_CASE

	__SYSTEM.TYPE_CLASS.TYPE_LTIME:
		_WriteInt(E_CustomTypes.eType_LTIME);
		_Copy(stArg.pValue, SIZEOF(LTIME));		
		
	ELSE
		F_InternalLog(
			E_LogLevel.eWarn,
			'FB_LogEntry.AddAnyArg',
			'Unhandled ANY type=%d',
			Tc2_Utilities.F_UDINT(stArg.TypeClass),
			Tc2_Utilities.EMPTY_ARG_VALUE,
			Tc2_Utilities.EMPTY_ARG_VALUE,
			Tc2_Utilities.EMPTY_ARG_VALUE
		);
		// TODO maybe rollback and ignore argument or use replacement value (null)
		bError := TRUE;
END_CASE

AddAnyArg := NOT bError;
END_METHOD

METHOD INTERNAL AddBuffer
VAR_INPUT
	pBuffer			: PVOID;
	nBufferLen		: UINT;
END_VAR
_Copy(pBuffer, nBufferLen);
END_METHOD

METHOD PUBLIC AddContext
VAR_INPUT
	eScope			: E_Scope;
	pBuffer			: PVOID;
	nBufferLen		: UINT;
END_VAR
_WriteByte(2); // Type 2: Context follows
_WriteByte(eScope);
_Copy(pBuffer, nBufferLen);
END_METHOD

METHOD INTERNAL AddTArg
VAR_INPUT
	nArgNo		: BYTE;
	stArg		: Tc2_Utilities.T_Arg;
END_VAR
IF bError THEN
	RETURN;
END_IF

IF stArg.eType = E_ArgType.ARGTYPE_UNKNOWN OR stArg.pData = 0 THEN
	RETURN;
END_IF

_WriteByte(1); // Type 1: Argument follows
_WriteByte(nArgNo);
_WriteInt(stArg.eType);

_Copy(ADR(stArg.eType), SIZEOF(stArg.eType));
CASE stArg.eType OF
	Tc2_Utilities.E_ArgType.ARGTYPE_BYTE:
		_Copy(stArg.pData, SIZEOF(BYTE));
	Tc2_Utilities.E_ArgType.ARGTYPE_WORD:
		_Copy(stArg.pData, SIZEOF(WORD));
	Tc2_Utilities.E_ArgType.ARGTYPE_DWORD:
		_Copy(stArg.pData, SIZEOF(DWORD));
	Tc2_Utilities.E_ArgType.ARGTYPE_REAL:
		_Copy(stArg.pData, SIZEOF(REAL));
	Tc2_Utilities.E_ArgType.ARGTYPE_LREAL:
		_Copy(stArg.pData, SIZEOF(LREAL));
	Tc2_Utilities.E_ArgType.ARGTYPE_SINT:
		_Copy(stArg.pData, SIZEOF(SINT));
	Tc2_Utilities.E_ArgType.ARGTYPE_INT:
		_Copy(stArg.pData, SIZEOF(INT));
	Tc2_Utilities.E_ArgType.ARGTYPE_DINT:
		_Copy(stArg.pData, SIZEOF(DINT));
	Tc2_Utilities.E_ArgType.ARGTYPE_USINT:
		_Copy(stArg.pData, SIZEOF(USINT));
	Tc2_Utilities.E_ArgType.ARGTYPE_UINT:
		_Copy(stArg.pData, SIZEOF(UINT));
	Tc2_Utilities.E_ArgType.ARGTYPE_UDINT:
		_Copy(stArg.pData, SIZEOF(UDINT));
	Tc2_Utilities.E_ArgType.ARGTYPE_STRING:
		_WriteString(stArg.pData);
	Tc2_Utilities.E_ArgType.ARGTYPE_BOOL:
		_WriteByte(SEL(Tc2_Utilities.PBOOL_TO_BOOL(stArg.pData), 0, 1));
	Tc2_Utilities.E_ArgType.ARGTYPE_ULARGE:
		_Copy(stArg.pData, SIZEOF(ULINT));
	Tc2_Utilities.E_ArgType.ARGTYPE_LARGE:
		_Copy(stArg.pData, SIZEOF(LINT));
	Tc2_Utilities.E_ArgType.ARGTYPE_LWORD:
		_Copy(stArg.pData, SIZEOF(LWORD));
END_CASE
END_METHOD

METHOD PUBLIC End : BOOL
VAR
	pWriteBuffer	: POINTER TO FB_LogBuffer;
	nBufferFree		: UINT;
	nActTaskIndex	: DINT;	
END_VAR
IF bError THEN
	RETURN;
END_IF

_WriteByte(255);

nActTaskIndex := GETCURTASKINDEXEX();

// end buffer write access
pWriteBuffer := PRG_TaskLog.TaskLogger.WriteBuffer;
IF pWriteBuffer^.BufferPtr <> pBuffer THEN 
	// sanity check
	F_InternalLog(
		E_LogLevel.eError,
		'FB_LogEntry.End',
		'Expected buffer to be the same.',
		Tc2_Utilities.EMPTY_ARG_VALUE,
		Tc2_Utilities.EMPTY_ARG_VALUE,
		Tc2_Utilities.EMPTY_ARG_VALUE,
		Tc2_Utilities.EMPTY_ARG_VALUE
	);
	
	bError := TRUE;
	
ELSIF pWriteBuffer^.BufferFree < nBufferCount THEN
	nBufferFree := pWriteBuffer^.BufferFree;
	F_InternalLog(
		E_LogLevel.eError,
		'FB_LogEntry.End',
		'Buffer capacity does not match buffer count. BufferFree=%d BufferCount=%d',
		Tc2_Utilities.F_UINT(nBufferFree),
		Tc2_Utilities.F_UINT(nBufferCount),
		Tc2_Utilities.EMPTY_ARG_VALUE,
		Tc2_Utilities.EMPTY_ARG_VALUE
	);

	bError := TRUE;
	
ELSE
	pWriteBuffer^.DataAdded(nBufferCount);	
END_IF

// Statistic
IF bError THEN
	IncUDINT(Log4TcInfo.aTaskInfo[nActTaskIndex].nAddLogToBufferErrorCount);
ELSE
	IncUDINT(Log4TcInfo.aTaskInfo[nActTaskIndex].nAddLogToBuffer);
END_IF

IF Log4TcInfo.aTaskInfo[nActTaskIndex].nMaxUsedBufferSize < pWriteBuffer^.BufferUsed THEN
	Log4TcInfo.aTaskInfo[nActTaskIndex].nMaxUsedBufferSize := pWriteBuffer^.BufferUsed;
END_IF

End := NOT bError;
END_METHOD

METHOD INTERNAL Start : BOOL
VAR_INPUT
	pLogger		: POINTER TO T_MaxString;
	pMessage		: POINTER TO T_MaxString;
	eLogLevel		: E_LogLevel;
	nTimeStampPlc	: LINT;
	nTimeStampClock	: LINT;
END_VAR
VAR
	fbSysTime		: Tc2_System.GETSYSTEMTIME;
	nTaskIndex		: DINT;
END_VAR
// Timestamp PLC
IF nTimestampPlc = 0 THEN
	fbSysTime();
	nTimeStampPlc := ULINT_TO_LINT(SHL(UDINT_TO_ULINT(fbSysTime.timeHiDW), 32) OR fbSysTime.timeLoDW);
END_IF

// Timestamp RTC
IF nTimestampClock = 0 THEN
	nTimestampClock := PRG_TaskLog.RtcTime;
END_IF

_Reset();

// Log-Entry Version
_WriteByte(1);

// Message
_WriteString(pMessage);

// Logger
_WriteString(pLogger);

// Level
_WriteUInt(eLogLevel);

// Timestamp PLC
_WriteLInt(nTimeStampPlc);

// Timestamp Clock
_WriteLInt(nTimeStampClock);

// Task Infos 
nTaskIndex := Tc2_System.GETCURTASKINDEXEX();
_WriteDInt(nTaskIndex);
_WriteString(ADR(TwinCAT_SystemInfoVarList._TaskInfo[nTaskIndex].TaskName));
_WriteUDInt(TwinCAT_SystemInfoVarList._TaskInfo[nTaskIndex].CycleCount);

// App Infos
_WriteString(ADR(TwinCAT_SystemInfoVarList._AppInfo.AppName));
_WriteString(ADR(TwinCAT_SystemInfoVarList._AppInfo.ProjectName));
_WriteUDInt(TwinCAT_SystemInfoVarList._AppInfo.OnlineChangeCnt);

Start := NOT bError;
END_METHOD

END_FUNCTION_BLOCK

// POUs/F_InternalLog
{attribute 'conditionalshow'}
FUNCTION INTERNAL F_InternalLog : BOOL
VAR_INPUT
	eLogLevel 			: E_LogLevel;
	sContext			: Tc2_System.T_MaxString;
	sMessageFmt			: Tc2_System.T_MaxString;
	stArg1				: Tc2_Utilities.T_Arg;
	stArg2				: Tc2_Utilities.T_Arg;
	stArg3				: Tc2_Utilities.T_Arg;
	stArg4				: Tc2_Utilities.T_Arg;
END_VAR
VAR
	sOutputStr			: T_MaxString;
	fbFormatStr			: FB_FormatString;
	aBoolToByte			: ARRAY[1..4] OF BYTE;
	pBool				: POINTER TO BOOL;
	nMask				: DWORD;
END_VAR

IF eLogLevel < Config.eInternalLog THEN
	RETURN;
END_IF

nMask := ADSLOG_MSGTYPE_LOG;

CASE eLogLevel OF
	E_LogLevel.eTrace:
		sOutputStr := '[TRACE] ';
	E_LogLevel.eDebug:
		sOutputStr := '[DEBUG] ';
	E_LogLevel.eInfo:
		sOutputStr := '[INFO] ';
		nMask := nMask OR ADSLOG_MSGTYPE_HINT;
	E_LogLevel.eWarn:
		sOutputStr := '[WARN] ';
		nMask := nMask OR ADSLOG_MSGTYPE_WARN;
	E_LogLevel.eError:
		sOutputStr := '[ERROR] ';
		nMask := nMask OR ADSLOG_MSGTYPE_ERROR;
	ELSE
		sOutputStr := '[FATAL] ';
		nMask := nMask OR ADSLOG_MSGTYPE_ERROR;
END_CASE

IF LEN(sContext) > 0 THEN
	sOutputStr := CONCAT(sOutputStr, CONCAT(sContext, ' - '));
END_IF

IF stArg1.eType = E_ArgType.ARGTYPE_BOOL THEN
	pBool := stArg1.pData;
	aBoolToByte[1] := SEL(pBool^, 0, 1);
	stArg1 := F_BYTE(aBoolToByte[1]);
END_IF

IF stArg2.eType = E_ArgType.ARGTYPE_BOOL THEN
	pBool := stArg2.pData;
	aBoolToByte[2] := SEL(pBool^, 0, 1);
	stArg2 := F_BYTE(aBoolToByte[2]);
END_IF

IF stArg3.eType = E_ArgType.ARGTYPE_BOOL THEN
	pBool := stArg3.pData;
	aBoolToByte[3] := SEL(pBool^, 0, 1);
	stArg3 := F_BYTE(aBoolToByte[3]);
END_IF

IF stArg4.eType = E_ArgType.ARGTYPE_BOOL THEN
	pBool := stArg4.pData;
	aBoolToByte[4] := SEL(pBool^, 0, 1);
	stArg4 := F_BYTE(aBoolToByte[4]);
END_IF


fbFormatStr(
	sFormat := sMessageFmt,
	arg1 	:= stArg1,
	arg2	:= stArg2,
	arg3	:= stArg3,
	arg4	:= stArg4,
);

sOutputStr := CONCAT(sOutputStr, fbFormatStr.sOut);

ADSLOGSTR(nMask, sOutputStr, '');

END_FUNCTION

// API/PRG_TaskLog
{attribute 'no_explicit_call' := 'no direct call necessary'}
PROGRAM PRG_TaskLog
VAR
	aTaskLogger			: ARRAY[1..SIZEOF(TwinCAT_SystemInfoVarList._TaskInfo)/SIZEOF(PlcTaskSystemInfo)] OF FB_Log4TcTask;
	aTaskRtcTime		: ARRAY[1..SIZEOF(TwinCAT_SystemInfoVarList._TaskInfo)/SIZEOF(PlcTaskSystemInfo)] OF FB_RTC_Sync;
END_VAR

(*
:Description: Sends collected log message of a single task to the service. 

This method must be called in each task which uses logging. It should be
called once a cycle.

**Example**

.. code:: 

    PRG_TaskLog.Call();
	
*)
METHOD PUBLIC Call
VAR
	nIdx	: DINT;
END_VAR
nIdx := Tc2_Utilities.GETCURTASKINDEXEX();
aTaskLogger[nIdx].Call();
aTaskRtcTime[nIdx].Call();
END_METHOD

(*
:Description: Initialise the task logger with custom parameter. 

This method must be called in each task which uses logging. As long as
the parameter do not change a single call is sufficient.

**Example**

.. code:: 

	IF _TaskInfo[GETCURTASKINDEXEX()].FirstCycle THEN
		// For Remote Log4TC Server change the AMS net ID and configure a route
	  PRG_TaskLog.Init('127.0.0.1.1.1');
	END_IF
    
*)
METHOD PUBLIC Init : BOOL
VAR_INPUT
	sAmsNetId	: Tc2_Utilities.T_AmsNetID;	(* The ams net id of the log service. Defaults to localhost (empty string). *)
END_VAR
aTaskLogger[Tc2_Utilities.GETCURTASKINDEXEX()].Init(sAmsNetId);
END_METHOD

PROPERTY INTERNAL RtcTime : LINT
GET
RtcTime := aTaskRtcTime[Tc2_Utilities.GETCURTASKINDEXEX()].RtcTime;
END_GET
END_PROPERTY

(*
:Description: Returns the ``I_ContextBuilder`` for task specific context
	properties. 

Task specific properties are added to each log message which is created
on the same task. 

For best performance properties should only be added or removed if the
values have changed.

**Example**

.. code:: 

	IF _TaskInfo[GETCURTASKINDEXEX()].FirstCycle THEN
		PRG_TaskLog.TaskContextBuilder.AddInt('machineNo', nMachineNumber);
	END_IF
    
*)
PROPERTY PUBLIC TaskContextBuilder : I_ContextBuilder
GET
TaskContextBuilder := aTaskLogger[GETCURTASKINDEXEX()].TaskContext;
END_GET
END_PROPERTY

PROPERTY INTERNAL TaskLogger : REFERENCE TO FB_Log4TcTask
GET
TaskLogger REF= aTaskLogger[GETCURTASKINDEXEX()];
END_GET
END_PROPERTY

END_PROGRAM

// POUs/FB_Log4TcTask
(*
Main code of Log4TC which manages log messages of a single task.
*)
{attribute 'no_explicit_call' := 'no direct call necessary'}
{attribute 'conditionalshow'}
FUNCTION_BLOCK INTERNAL FB_Log4TcTask
VAR CONSTANT
	nAdsPort			: UINT := 16150; 
	nLogIndexGrp		: UINT := 1;
	nLogIndexOffs		: UINT := 1;	
END_VAR
VAR
	nTaskIndex			: DINT;
	fbTaskContext		: FB_ContextBuilder;
	sAmsNetId			: Tc2_System.T_AmsNetID := '';
	
	nWriteBuffer		: UINT (1..2) := 1;
	fbLogBuffer1		: FB_LogBuffer;
	fbLogBuffer2		: FB_LogBuffer;
END_VAR

METHOD PRIVATE _InitAndCheckTask : BOOL
VAR
	nActTaskIndex		: DINT;
END_VAR
_InitAndCheckTask := TRUE;

nActTaskIndex := Tc2_System.GETCURTASKINDEXEX();
IF nTaskIndex = 0 AND nActTaskIndex > 0 THEN
	nTaskIndex := nActTaskIndex;
ELSIF nTaskIndex <> nActTaskIndex OR nActTaskIndex = 0 THEN
	F_InternalLog(
		E_LogLevel.eFatal,
		'Log4TcTask._InitAndCheckTask',
		'Log4Tc called in wrong task (expected=%d actual=%d)',
		F_DINT(nTaskIndex),
		F_DINT(nActTaskIndex),
		Tc2_Utilities.EMPTY_ARG_VALUE,
		Tc2_Utilities.EMPTY_ARG_VALUE
	);
	_InitAndCheckTask := FALSE;
END_IF
END_METHOD

PROPERTY PRIVATE _ReadBuffer : POINTER TO FB_LogBuffer
GET
IF nWriteBuffer = 1 THEN
	_ReadBuffer := ADR(fbLogBuffer2);
ELSE
	_ReadBuffer := ADR(fbLogBuffer1);
END_IF
END_GET
END_PROPERTY

(*
Should be called regularly in the same task as its instance was
declared.
*)
METHOD INTERNAL Call
VAR
	pWriteBuffer		: POINTER TO FB_LogBuffer;
	pReadBuffer			: POINTER TO FB_LogBuffer;
END_VAR
VAR_INST
	nState				: UINT;
	fbAdsWriteMsg		: Tc2_System.ADSWRITE:=(PORT:=nAdsPort);
	fbRetryWait			: Tc2_System.TON:=(PT:=T#5S);
END_VAR
IF NOT _InitAndCheckTask() THEN
	RETURN;
END_IF

CASE nState OF
	0: // Init
		nState := 10;
		
	10: // Wait for log entry; add them to the send buffer
		pWriteBuffer := WriteBuffer;

		IF pWriteBuffer^.BufferUsed > 0 THEN
			// Switch buffer for next write
			nWriteBuffer := SEL(nWriteBuffer = 1, 1 , 2);
			
			fbAdsWriteMsg(WRITE:=FALSE);
			fbAdsWriteMsg(
				WRITE	:= TRUE,
				NETID	:= sAmsNetId,
				IDXGRP 	:= nLogIndexGrp,
				IDXOFFS := nLogIndexOffs,
				LEN		:= pWriteBuffer^.BufferUsed,
				SRCADDR	:= pWriteBuffer^.BufferStartPtr,
			);
			
			F_InternalLog(
				E_LogLevel.eDebug,
				'FB_Log4TcTask.Call',
				'Sending message with size %d.',
				Tc2_Utilities.F_UDINT(fbAdsWriteMsg.LEN),
				Tc2_Utilities.EMPTY_ARG_VALUE,
				Tc2_Utilities.EMPTY_ARG_VALUE,
				Tc2_Utilities.EMPTY_ARG_VALUE
			);				
		
			nState := 20;			
		END_IF		
		
	20: // Wait for sent data
		fbAdsWriteMsg();
		IF NOT fbAdsWriteMsg.BUSY THEN
			IF fbAdsWriteMsg.ERR THEN
				F_InternalLog(
					E_LogLevel.eFatal,
					'Log4TcTask.Call',
					'Error sending log message to handler. task=%d adsErrId=%d',
					F_DINT(nTaskIndex),
					F_UDINT(fbAdsWriteMsg.ERRID),
					Tc2_Utilities.EMPTY_ARG_VALUE,
					Tc2_Utilities.EMPTY_ARG_VALUE
				);
				
				IncUDINT(Log4TcInfo.aTaskInfo[nTaskIndex].nSendLogBufferErrorCount);
				
				fbRetryWait(IN:=FALSE);
				nState := 30;
			ELSE
				F_InternalLog(
					E_LogLevel.eDebug,
					'FB_Log4TcTask.Call',
					'Message successfully sent.',
					Tc2_Utilities.EMPTY_ARG_VALUE,
					Tc2_Utilities.EMPTY_ARG_VALUE,
					Tc2_Utilities.EMPTY_ARG_VALUE,
					Tc2_Utilities.EMPTY_ARG_VALUE
				);	
				
				pReadBuffer := _ReadBuffer;
				pReadBuffer^.Clear();
				nState := 10;
			END_IF
		END_IF
		
	30: // Retry wait sending
		fbRetryWait(IN:=TRUE);
		IF fbRetryWait.Q THEN
			// sending same data again
			fbAdsWriteMsg(WRITE:=FALSE);
			fbAdsWriteMsg(WRITE:=TRUE);
			nState := 20;
		END_IF
	
END_CASE
END_METHOD

METHOD INTERNAL Init
VAR_INPUT
	sAmsNetId	: Tc2_Utilities.T_AmsNetID;
END_VAR
THIS^.sAmsNetId := sAmsNetId;
END_METHOD

PROPERTY INTERNAL TaskContext : REFERENCE TO FB_ContextBuilder
GET
TaskContext REF= fbTaskContext;
END_GET
END_PROPERTY

PROPERTY INTERNAL WriteBuffer : POINTER TO FB_LogBuffer
GET
IF nWriteBuffer = 1 THEN
	WriteBuffer := ADR(fbLogBuffer1);
ELSE
	WriteBuffer := ADR(fbLogBuffer2);
END_IF
END_GET
END_PROPERTY

END_FUNCTION_BLOCK

// POUs/Utils/FB_LogBuffer
{attribute 'no_explicit_call' := 'no direct call necessary'}
FUNCTION_BLOCK INTERNAL FB_LogBuffer
VAR
	aBuffer			: ARRAY[1..Config.nBufferLen] OF BYTE;
	nBufferCount	: UINT;
END_VAR

PROPERTY INTERNAL BufferFree : UINT
GET
BufferFree := Config.nBufferLen - nBufferCount;
END_GET
END_PROPERTY

PROPERTY INTERNAL BufferPtr : PVOID
GET
BufferPtr := ADR(aBuffer) + nBufferCount;
END_GET
END_PROPERTY

PROPERTY INTERNAL BufferStartPtr : PVOID
GET
BufferStartPtr := ADR(aBuffer);
END_GET
END_PROPERTY

PROPERTY INTERNAL BufferUsed : UINT
GET
BufferUsed := nBufferCount;
END_GET
END_PROPERTY

METHOD INTERNAL Clear
nBufferCount := 0;
END_METHOD

METHOD INTERNAL DataAdded 
VAR_INPUT
	nNewData		: UINT;
END_VAR
nBufferCount := nBufferCount + nNewData;
IF nBufferCount > Config.nBufferLen THEN
	F_InternalLog(
		E_LogLevel.eError,
		'FB_LogBuffer.DataAdded',
		'Buffer overflow adding to log buffer.',
		Tc2_Utilities.EMPTY_ARG_VALUE,
		Tc2_Utilities.EMPTY_ARG_VALUE,
		Tc2_Utilities.EMPTY_ARG_VALUE,
		Tc2_Utilities.EMPTY_ARG_VALUE
	);
END_IF
END_METHOD

END_FUNCTION_BLOCK

// POUs/Utils/IncUDINT
FUNCTION INTERNAL IncUDINT : UDINT
VAR_INPUT
	refValue		: REFERENCE TO UDINT;
END_VAR

IncUDINT := (refValue := refValue + 1);

END_FUNCTION

// POUs/Utils/FB_RTC_Sync
FUNCTION_BLOCK INTERNAL FB_RTC_Sync
VAR
	fbRtcEx2		: Tc2_Utilities.RTC_EX2;
END_VAR

METHOD INTERNAL Call : BOOL
VAR_INPUT
END_VAR
VAR_INST
	fbGetTime		: Tc2_Utilities.NT_GetTime;
	fbSyncTimer		: Tc2_Standard.TON := (PT:=T#10M);
	bInit			: BOOL;	
END_VAR
fbSyncTimer(IN:=NOT fbSyncTimer.Q);

fbGetTime.START S= fbSyncTimer.Q OR NOT bInit;
fbGetTime();

IF NOT fbGetTime.BUSY THEN
	fbGetTime.START := FALSE;
	IF NOT fbGetTime.ERR THEN
		fbRtcEx2.PDT := fbGetTime.TIMESTR;
		fbRtcEx2.EN := TRUE;
		fbRtcEx2.PMICRO := 0;
	END_IF
END_IF

fbRtcEx2();
fbRtcEx2.EN := FALSE;

bInit := TRUE;
END_METHOD

PROPERTY INTERNAL RtcTime : LINT
GET
VAR
	nFileTime	: Tc2_Utilities.T_FILETIME;
END_VAR
fbRtcEx2();
IF fbRtcEx2.Q THEN
	nFileTime := Tc2_Utilities.SYSTEMTIME_TO_FILETIME(fbRtcEx2.CDT);
	RtcTime := ULINT_TO_LINT(SHL(UDINT_TO_ULINT(nFileTime.dwHighDateTime), 32) OR nFileTime.dwLowDateTime)
		+ fbRtcEx2.CMICRO * LINT#10;
ELSE
	Rtctime := 0;
END_IF
END_GET
END_PROPERTY

END_FUNCTION_BLOCK

// API/Context/FB_ScopedContext
(*
:Description: Provide nested scoped context properties. 

This function block can be used to define context properties, which
are valid from ``Begin()`` to ``End()``. This context properties can
be used to provide call-stack specific properties for example when
using multi-instance.

The maximum nested level can be configured with ``Config.nMaxScopedContext``.
The default level is 4.

**Example**

.. code:: 

	fbMachine1Ctx	: FB_ScopedContext;
	fbMachine2Ctx	: FB_ScopedContext;
	
	IF bInit THEN
		fbMachine1Ctx.ContextBuilder.AddInt('MachineNo', 1);
		fbMachine2Ctx.ContextBuilder.AddInt('MachineNo', 2);
	END_IF
	
    fbMachine1Ctx.Begin();
	// Call code for machine 1
	fbMachine1Ctx.End();
	
    fbMachine2Ctx.Begin();
	// Call code for machine 2
	fbMachine2Ctx.End();
*)
{attribute 'no_explicit_call' := 'no direct call necessary'}
FUNCTION_BLOCK PUBLIC FB_ScopedContext
VAR
	fbContext			: FB_ContextBuilder;
	bActive				: BOOL;
END_VAR

(*
:Description: Begins a nested context. 

Each ``Begin()`` call must be balance by an ``End()`` call in the same
order if nested context are used.
*)
METHOD PUBLIC Begin
VAR
	refTaskContextStack		: REFERENCE TO ST_ScopedContextStack;
END_VAR
IF NOT bActive THEN
	bActive := TRUE;
	
	refTaskContextStack REF= PRG_ScopedContextStack.TaskContextStack;
	
	IF refTaskContextStack.nScopeContextCount < Config.nMaxScopedContext THEN
		refTaskContextStack.aScopedContext[refTaskContextStack.nScopeContextCount] := fbContext;
		refTaskContextStack.nScopeContextCount := refTaskContextStack.nScopeContextCount + 1;
	ELSE
		F_InternalLog(
			E_LogLevel.eError,
			'FB_ScopedContext.Begin',
			'Too many nested scoped context.',
			Tc2_Utilities.EMPTY_ARG_VALUE,
			Tc2_Utilities.EMPTY_ARG_VALUE,
			Tc2_Utilities.EMPTY_ARG_VALUE,
			Tc2_Utilities.EMPTY_ARG_VALUE
		);
	END_IF
ELSE
	F_InternalLog(
		E_LogLevel.eError,
		'FB_ScopedContext.Begin',
		'Begin() called twice without End()',
		Tc2_Utilities.EMPTY_ARG_VALUE,
		Tc2_Utilities.EMPTY_ARG_VALUE,
		Tc2_Utilities.EMPTY_ARG_VALUE,
		Tc2_Utilities.EMPTY_ARG_VALUE
	);
END_IF
END_METHOD

(*
:Description: Returns the context builder for this scoped context. 

For best performance the context build should only be called on
changed values.
*)
PROPERTY PUBLIC ContextBuilder : I_ContextBuilder
GET
ContextBuilder := fbContext;
END_GET
END_PROPERTY

(*
:Description: Ends a nested context. 

Each ``Begin()`` call must be balance by an ``End()`` call in the same
order if nested context are used.
*)
METHOD PUBLIC End
VAR
	nIdx					: INT;
	refTaskContextStack		: REFERENCE TO ST_ScopedContextStack;
	iThisContextBuilder		: I_ContextBuilder;
END_VAR
IF bActive THEN
	bActive := FALSE;
	
	refTaskContextStack REF= PRG_ScopedContextStack.TaskContextStack;
	iThisContextBuilder := fbContext;
	
	// expected at top
	IF refTaskContextStack.nScopeContextCount > 0 
			AND_THEN refTaskContextStack.aScopedContext[refTaskContextStack.nScopeContextCount - 1] = iThisContextBuilder 
	THEN
		refTaskContextStack.nScopeContextCount := refTaskContextStack.nScopeContextCount - 1;
		RETURN;
	END_IF
	
	// try to find it in the stack
	FOR nIdx := UINT_TO_INT(refTaskContextStack.nScopeContextCount) - 1 TO 0 BY -1 DO
		IF refTaskContextStack.aScopedContext[nIdx] = iThisContextBuilder THEN
			F_InternalLog(
				E_LogLevel.eError,
				'FB_ScopedContext.End',
				'Removed scoped context at %d instead of %d-1 - ensure Begin/End are called in order.',
				Tc2_Utilities.F_INT(nIdx),
				Tc2_Utilities.F_UINT(refTaskContextStack.nScopeContextCount),
				Tc2_Utilities.EMPTY_ARG_VALUE,
				Tc2_Utilities.EMPTY_ARG_VALUE
			);	
		
			refTaskContextStack.nScopeContextCount := INT_TO_UINT(nIdx);
			RETURN;
		END_IF
	END_FOR
	
	F_InternalLog(
		E_LogLevel.eError,
		'FB_ScopedContext.End',
		'Cannot remove non existing scope',
		Tc2_Utilities.EMPTY_ARG_VALUE,
		Tc2_Utilities.EMPTY_ARG_VALUE,
		Tc2_Utilities.EMPTY_ARG_VALUE,
		Tc2_Utilities.EMPTY_ARG_VALUE
	);	
ELSE
	F_InternalLog(
		E_LogLevel.eError,
		'FB_ScopedContext.End',
		'End() called without Begin()',
		Tc2_Utilities.EMPTY_ARG_VALUE,
		Tc2_Utilities.EMPTY_ARG_VALUE,
		Tc2_Utilities.EMPTY_ARG_VALUE,
		Tc2_Utilities.EMPTY_ARG_VALUE
	);
END_IF
END_METHOD

END_FUNCTION_BLOCK

// POUs/PRG_ScopedContextStack
{attribute 'conditionalshow'}
PROGRAM INTERNAL PRG_ScopedContextStack
VAR
	aContextStack		: ARRAY[1..SIZEOF(TwinCAT_SystemInfoVarList._TaskInfo)/SIZEOF(PlcTaskSystemInfo)] OF ST_ScopedContextStack;
END_VAR

PROPERTY INTERNAL TaskContextStack : REFERENCE TO ST_ScopedContextStack
GET
VAR
	nTaskIdx	: DINT;
END_VAR
nTaskIdx := Tc2_System.GETCURTASKINDEXEX();
TaskContextStack REF= aContextStack[nTaskIdx];
END_GET
END_PROPERTY

END_PROGRAM

// API/Full/FB_LoggerLAC
(*
:Description: Writes log messages with the same logger and context. 

This function block allows to log messages with the same logger and
context without repeating the data on each log call.


The logger must be specified during instantiation. If the
constant `Const.sLoggerFromInstance` is specified, then the logger is 
retrieved from the instance path of the FB (only possible with 
instantiation in FBs).

**Example**

.. code:: 
    VAR
        fbLog   : FB_LoggerLAC(Const.sLoggerFromInstance);
    END_VAR

	fbLog(
		eLogLevel 	:= E_LogLevel.eInfo,
		sMessage 	:= 'Something happens with code {code}',
		aArg1 		:= nCode
	);
	
*)
{attribute 'reflection'} 
FUNCTION_BLOCK FB_LoggerLAC
VAR_INPUT
	bExecute			: BOOL := TRUE;
	eLogLevel			: E_LogLevel;
	sMessage			: Tc2_System.T_MaxString;
	aArg1				: ANY;
	aArg2				: ANY;
	aArg3				: ANY;
	aArg4				: ANY;
	aArg5				: ANY;	
	aArg6				: ANY;	
	aArg7				: ANY;	
	aArg8				: ANY;	
	aArg9				: ANY;	
	aArg10				: ANY;	
	iContextBuilder		: I_ContextBuilder := 0;	
END_VAR
VAR
    {attribute 'instance-path'} 
    {attribute 'noinit'} // 'log4tc.log4Tc_Tester.MAIN.fbLog' bwz. 'log4tc.log4Tc_Tester.GVL.fbLog'
    sInstancePath		: T_MaxString; 	
	sLogger				: T_MaxString;	// Initialized from FB_init	
	bInitLogger			: BOOL;
	fbLoggerContext		: FB_ContextBuilder;	// Logger scoped context
END_VAR
VAR_TEMP
	fbLogEntry			: FB_LogEntry();
	iLogEntryAdder		: I_LogEntryAdder;
	nIdx				: UINT;
	nFindIdx			: INT;
	refScopedContext	: REFERENCE TO ST_ScopedContextStack;
	pBuffer				: PVOID;
	nBufferCount		: UINT;	
END_VAR

IF bExecute THEN
	IF NOT bInitLogger THEN
		bInitLogger := TRUE;
		IF sLogger = Const.sLoggerFromInstance THEN
			// strip application/project from instance path
			nFindIdx := Tc2_Standard.FIND(sInstancePath, '.');
			IF nFindIdx > 0 THEN
				sInstancePath := Tc2_Standard.DELETE(sInstancePath, nFindIdx + 1, 0);
				nFindIdx := Tc2_Standard.FIND(sInstancePath, '.');
				IF nFindIdx > 0 THEN
					sInstancePath := Tc2_Standard.DELETE(sInstancePath, nFindIdx + 1, 0);
					sLogger := sInstancePath;
				END_IF
			END_IF
		END_IF
	END_IF	

	fbLogEntry.Start(
		pLogger			:= ADR(sLogger),
		pMessage		:= ADR(sMessage),
		eLogLevel		:= eLogLevel,
		nTimeStampPlc	:= 0,
		nTimeStampClock	:= 0
	);
	
	fbLogEntry.AddAnyArg(1, aArg1);
	fbLogEntry.AddAnyArg(2, aArg2);
	fbLogEntry.AddAnyArg(3, aArg3);
	fbLogEntry.AddAnyArg(4, aArg4);
	fbLogEntry.AddAnyArg(5, aArg5);
	fbLogEntry.AddAnyArg(6, aArg6);
	fbLogEntry.AddAnyArg(7, aArg7);
	fbLogEntry.AddAnyArg(8, aArg8);
	fbLogEntry.AddAnyArg(9, aArg9);
	fbLogEntry.AddAnyArg(10, aArg10);
	
	IF __QUERYINTERFACE(PRG_TaskLog.TaskLogger.TaskContext, iLogEntryAdder) THEN
		iLogEntryAdder.AddToLogEntry(E_Scope.eTask, fbLogEntry);
	END_IF
	
	refScopedContext REF= PRG_ScopedContextStack.TaskContextStack;
	FOR nIdx := 0 TO refScopedContext.nScopeContextCount - 1 DO
		IF __QUERYINTERFACE(refScopedContext.aScopedContext[nIdx], iLogEntryAdder) THEN
			iLogEntryAdder.AddToLogEntry(E_Scope.eScoped, fbLogEntry);
		END_IF
	END_FOR
	
	fbLoggerContext.AddToLogEntry(E_Scope.eLogger, fbLogEntry);
	
	IF iContextBuilder <> 0 AND __QUERYINTERFACE(iContextBuilder, iLogEntryAdder) THEN
		iLogEntryAdder.AddToLogEntry(E_Scope.eLog, fbLogEntry);
	END_IF
	
	fbLogEntry.End();
END_IF

// reset arguments to default values
bExecute := TRUE;
aArg1.pValue := 
	aArg2.pValue := 
	aArg3.pValue := 
	aArg4.pValue := 
	aArg5.pValue := 
	aArg6.pValue := 
	aArg7.pValue := 
	aArg8.pValue := 
	aArg9.pValue := 
	aArg10.pValue := 0;
aArg1.TypeClass :=
	aArg2.TypeClass :=
	aArg3.TypeClass :=
	aArg4.TypeClass :=
	aArg5.TypeClass :=
	aArg6.TypeClass :=
	aArg7.TypeClass :=
	aArg8.TypeClass :=
	aArg9.TypeClass :=
	aArg10.TypeClass := __SYSTEM.TYPE_CLASS.TYPE_NONE;
iContextBuilder := 0;

METHOD FB_init : BOOL
VAR_INPUT
	bInitRetains : BOOL; // if TRUE, the retain variables are initialized (warm start / cold start)
	bInCopyCode : BOOL;  // if TRUE, the instance afterwards gets moved into the copy code (online change)
	sLogger		: T_MaxString;
END_VAR
THIS^.sLogger := sLogger;
END_METHOD

PROPERTY PUBLIC LoggerContext : I_ContextBuilder
GET
LoggerContext := fbLoggerContext;
END_GET
END_PROPERTY

END_FUNCTION_BLOCK

// API/Simple/Any/F_LogA1
FUNCTION F_LogA1 
VAR_INPUT
	eLogLevel		: E_LogLevel;
	sMessage		: T_MaxString;
	aArg1			: ANY;
END_VAR

F_LogLA1(eLogLevel, Const.sGlobalLogger, sMessage, aArg1);

END_FUNCTION

// API/Simple/Any/F_LogLA1
FUNCTION F_LogLA1 
VAR_INPUT
	eLogLevel		: E_LogLevel;
	sLogger			: T_MaxString;
	sMessage		: T_MaxString;
	aArg1			: ANY;
END_VAR
VAR 
	aEmptyArg		: BYTE;
END_VAR

F_LogA(
	eLogLevel,
	sLogger,
	sMessage,
	1,
	aArg1,
	aEmptyArg,
	aEmptyArg,
	aEmptyArg,
	aEmptyArg,
	aEmptyArg,
	aEmptyArg,
	aEmptyArg,
	aEmptyArg,
	aEmptyArg,
	0
);

END_FUNCTION

// POUs/F_LogA
{attribute 'conditionalshow'}
FUNCTION INTERNAL F_LogA 
VAR_INPUT
	eLogLevel		: E_LogLevel;
	sLogger			: T_MaxString;
	sMessage		: T_MaxString;
	nArgCount		: UINT (0..10);
	aArg1			: ANY;
	aArg2			: ANY;
	aArg3			: ANY;
	aArg4			: ANY;
	aArg5			: ANY;
	aArg6			: ANY;
	aArg7			: ANY;
	aArg8			: ANY;
	aArg9			: ANY;
	aArg10			: ANY;
	iContextBuilder	: I_ContextBuilder;
END_VAR
VAR
	fbLogEntry			: FB_LogEntry();
	pBuffer				: PVOID;
	nBufferCount		: UINT;	
	iLogEntryAdder		: I_LogEntryAdder;
	nIdx				: UINT;
	refScopedContext	: REFERENCE TO ST_ScopedContextStack;
END_VAR

fbLogEntry.Start(
	pLogger			:= ADR(sLogger),
	pMessage		:= ADR(sMessage),
	eLogLevel		:= eLogLevel,
	nTimeStampPlc	:= 0,
	nTimeStampClock	:= 0
);

IF nArgCount >= 1 THEN
	fbLogEntry.AddAnyArg(1, aArg1);
END_IF
IF nArgCount >= 2 THEN 
	fbLogEntry.AddAnyArg(2, aArg2);
END_IF
IF nArgCount >= 3 THEN 
	fbLogEntry.AddAnyArg(3, aArg3);
END_IF
IF nArgCount >= 4 THEN 
	fbLogEntry.AddAnyArg(4, aArg4);
END_IF
IF nArgCount >= 5 THEN 
	fbLogEntry.AddAnyArg(5, aArg5);
END_IF
IF nArgCount >= 6 THEN 
	fbLogEntry.AddAnyArg(6, aArg6);
END_IF
IF nArgCount >= 7 THEN 
	fbLogEntry.AddAnyArg(7, aArg7);
END_IF
IF nArgCount >= 8 THEN 
	fbLogEntry.AddAnyArg(8, aArg8);
END_IF
IF nArgCount >= 9 THEN 
	fbLogEntry.AddAnyArg(9, aArg9);
END_IF
IF nArgCount >= 10 THEN 
	fbLogEntry.AddAnyArg(10, aArg10);
END_IF

IF __QUERYINTERFACE(PRG_TaskLog.TaskLogger.TaskContext, iLogEntryAdder) THEN
	iLogEntryAdder.AddToLogEntry(E_Scope.eTask, fbLogEntry);
END_IF

refScopedContext REF= PRG_ScopedContextStack.TaskContextStack;
IF refScopedContext.nScopeContextCount > 0 THEN
	FOR nIdx := 0 TO refScopedContext.nScopeContextCount - 1 DO
		IF __QUERYINTERFACE(refScopedContext.aScopedContext[nIdx], iLogEntryAdder) THEN
			iLogEntryAdder.AddToLogEntry(E_Scope.eScoped, fbLogEntry);
		END_IF
	END_FOR
END_IF

IF iContextBuilder <> 0 AND __QUERYINTERFACE(iContextBuilder, iLogEntryAdder) THEN
	iLogEntryAdder.AddToLogEntry(E_Scope.eLogger, fbLogEntry);
END_IF

fbLogEntry.End();

END_FUNCTION

// API/Simple/Any/F_LogA10
FUNCTION F_LogA10 
VAR_INPUT
	eLogLevel		: E_LogLevel;
	sMessage		: T_MaxString;
	aArg1			: ANY;
	aArg2			: ANY;
	aArg3			: ANY;
	aArg4			: ANY;
	aArg5			: ANY;
	aArg6			: ANY;
	aArg7			: ANY;
	aArg8			: ANY;
	aArg9			: ANY;
	aArg10			: ANY;
END_VAR

F_LogLA10(eLogLevel, Const.sGlobalLogger, sMessage, aArg1, aArg2, aArg3, aArg4, aArg5, aArg6, aArg7, aArg8, aArg9, aArg10);

END_FUNCTION

// API/Simple/Any/F_LogLA10
FUNCTION F_LogLA10 
VAR_INPUT
	eLogLevel		: E_LogLevel;
	sLogger			: T_MaxString;
	sMessage		: T_MaxString;
	aArg1			: ANY;
	aArg2			: ANY;
	aArg3			: ANY;
	aArg4			: ANY;
	aArg5			: ANY;
	aArg6			: ANY;
	aArg7			: ANY;
	aArg8			: ANY;
	aArg9			: ANY;
	aArg10			: ANY;
END_VAR

F_LogA(
	eLogLevel,
	sLogger,
	sMessage,
	10,
	aArg1,
	aArg2,
	aArg3,
	aArg4,
	aArg5,
	aArg6,
	aArg7,
	aArg8,
	aArg9,
	aArg10,
	0
);

END_FUNCTION

// API/Simple/Any/F_LogA2
FUNCTION F_LogA2 
VAR_INPUT
	eLogLevel		: E_LogLevel;
	sMessage		: T_MaxString;
	aArg1			: ANY;
	aArg2			: ANY;
END_VAR

F_LogLA2(eLogLevel, Const.sGlobalLogger, sMessage, aArg1, aArg2);

END_FUNCTION

// API/Simple/Any/F_LogLA2
FUNCTION F_LogLA2 
VAR_INPUT
	eLogLevel		: E_LogLevel;
	sLogger			: T_MaxString;
	sMessage		: T_MaxString;
	aArg1			: ANY;
	aArg2			: ANY;
END_VAR
VAR 
	aEmptyArg		: BYTE;
END_VAR

F_LogA(
	eLogLevel,
	sLogger,
	sMessage,
	2,
	aArg1,
	aArg2,
	aEmptyArg,
	aEmptyArg,
	aEmptyArg,
	aEmptyArg,
	aEmptyArg,
	aEmptyArg,
	aEmptyArg,
	aEmptyArg,
	0
);

END_FUNCTION

// API/Simple/Any/F_LogA3
FUNCTION F_LogA3 
VAR_INPUT
	eLogLevel		: E_LogLevel;
	sMessage		: T_MaxString;
	aArg1			: ANY;
	aArg2			: ANY;
	aArg3			: ANY;
END_VAR

F_LogLA3(eLogLevel, Const.sGlobalLogger, sMessage, aArg1, aArg2, aArg3);

END_FUNCTION

// API/Simple/Any/F_LogLA3
FUNCTION F_LogLA3 
VAR_INPUT
	eLogLevel		: E_LogLevel;
	sLogger			: T_MaxString;
	sMessage		: T_MaxString;
	aArg1			: ANY;
	aArg2			: ANY;
	aArg3			: ANY;
END_VAR
VAR 
	aEmptyArg		: BYTE;
END_VAR

F_LogA(
	eLogLevel,
	sLogger,
	sMessage,
	3,
	aArg1,
	aArg2,
	aArg3,
	aEmptyArg,
	aEmptyArg,
	aEmptyArg,
	aEmptyArg,
	aEmptyArg,
	aEmptyArg,
	aEmptyArg,
	0
);

END_FUNCTION

// API/Simple/Any/F_LogA4
FUNCTION F_LogA4 
VAR_INPUT
	eLogLevel		: E_LogLevel;
	sMessage		: T_MaxString;
	aArg1			: ANY;
	aArg2			: ANY;
	aArg3			: ANY;
	aArg4			: ANY;
END_VAR

F_LogLA4(eLogLevel, Const.sGlobalLogger, sMessage, aArg1, aArg2, aArg3, aArg4);

END_FUNCTION

// API/Simple/Any/F_LogLA4
FUNCTION F_LogLA4 
VAR_INPUT
	eLogLevel		: E_LogLevel;
	sLogger			: T_MaxString;
	sMessage		: T_MaxString;
	aArg1			: ANY;
	aArg2			: ANY;
	aArg3			: ANY;
	aArg4			: ANY;
END_VAR
VAR 
	aEmptyArg		: BYTE;
END_VAR

F_LogA(
	eLogLevel,
	sLogger,
	sMessage,
	4,
	aArg1,
	aArg2,
	aArg3,
	aArg4,
	aEmptyArg,
	aEmptyArg,
	aEmptyArg,
	aEmptyArg,
	aEmptyArg,
	aEmptyArg,
	0
);

END_FUNCTION

// API/Simple/Any/F_LogA5
FUNCTION F_LogA5 
VAR_INPUT
	eLogLevel		: E_LogLevel;
	sMessage		: T_MaxString;
	aArg1			: ANY;
	aArg2			: ANY;
	aArg3			: ANY;
	aArg4			: ANY;
	aArg5			: ANY;
END_VAR

F_LogLA5(eLogLevel, Const.sGlobalLogger, sMessage, aArg1, aArg2, aArg3, aArg4, aArg5);

END_FUNCTION

// API/Simple/Any/F_LogLA5
FUNCTION F_LogLA5 
VAR_INPUT
	eLogLevel		: E_LogLevel;
	sLogger			: T_MaxString;
	sMessage		: T_MaxString;
	aArg1			: ANY;
	aArg2			: ANY;
	aArg3			: ANY;
	aArg4			: ANY;
	aArg5			: ANY;
END_VAR
VAR 
	aEmptyArg		: BYTE;
END_VAR

F_LogA(
	eLogLevel,
	sLogger,
	sMessage,
	5,
	aArg1,
	aArg2,
	aArg3,
	aArg4,
	aArg5,
	aEmptyArg,
	aEmptyArg,
	aEmptyArg,
	aEmptyArg,
	aEmptyArg,
	0
);

END_FUNCTION

// API/Simple/Any/F_LogA6
FUNCTION F_LogA6 
VAR_INPUT
	eLogLevel		: E_LogLevel;
	sMessage		: T_MaxString;
	aArg1			: ANY;
	aArg2			: ANY;
	aArg3			: ANY;
	aArg4			: ANY;
	aArg5			: ANY;
	aArg6			: ANY;
END_VAR

F_LogLA6(eLogLevel, Const.sGlobalLogger, sMessage, aArg1, aArg2, aArg3, aArg4, aArg5, aArg6);

END_FUNCTION

// API/Simple/Any/F_LogLA6
FUNCTION F_LogLA6 
VAR_INPUT
	eLogLevel		: E_LogLevel;
	sLogger			: T_MaxString;
	sMessage		: T_MaxString;
	aArg1			: ANY;
	aArg2			: ANY;
	aArg3			: ANY;
	aArg4			: ANY;
	aArg5			: ANY;
	aArg6			: ANY;
END_VAR
VAR 
	aEmptyArg		: BYTE;
END_VAR

F_LogA(
	eLogLevel,
	sLogger,
	sMessage,
	6,
	aArg1,
	aArg2,
	aArg3,
	aArg4,
	aArg5,
	aArg6,
	aEmptyArg,
	aEmptyArg,
	aEmptyArg,
	aEmptyArg,
	0
);

END_FUNCTION

// API/Simple/Any/F_LogA7
FUNCTION F_LogA7 
VAR_INPUT
	eLogLevel		: E_LogLevel;
	sMessage		: T_MaxString;
	aArg1			: ANY;
	aArg2			: ANY;
	aArg3			: ANY;
	aArg4			: ANY;
	aArg5			: ANY;
	aArg6			: ANY;
	aArg7			: ANY;
END_VAR

F_LogLA7(eLogLevel, Const.sGlobalLogger, sMessage, aArg1, aArg2, aArg3, aArg4, aArg5, aArg6, aArg7);

END_FUNCTION

// API/Simple/Any/F_LogLA7
FUNCTION F_LogLA7 
VAR_INPUT
	eLogLevel		: E_LogLevel;
	sLogger			: T_MaxString;
	sMessage		: T_MaxString;
	aArg1			: ANY;
	aArg2			: ANY;
	aArg3			: ANY;
	aArg4			: ANY;
	aArg5			: ANY;
	aArg6			: ANY;
	aArg7			: ANY;
END_VAR
VAR 
	aEmptyArg		: BYTE;
END_VAR

F_LogA(
	eLogLevel,
	sLogger,
	sMessage,
	7,
	aArg1,
	aArg2,
	aArg3,
	aArg4,
	aArg5,
	aArg6,
	aArg7,
	aEmptyArg,
	aEmptyArg,
	aEmptyArg,
	0
);

END_FUNCTION

// API/Simple/Any/F_LogA8
FUNCTION F_LogA8 
VAR_INPUT
	eLogLevel		: E_LogLevel;
	sMessage		: T_MaxString;
	aArg1			: ANY;
	aArg2			: ANY;
	aArg3			: ANY;
	aArg4			: ANY;
	aArg5			: ANY;
	aArg6			: ANY;
	aArg7			: ANY;
	aArg8			: ANY;
END_VAR

F_LogLA8(eLogLevel, Const.sGlobalLogger, sMessage, aArg1, aArg2, aArg3, aArg4, aArg5, aArg6, aArg7, aArg8);

END_FUNCTION

// API/Simple/Any/F_LogLA8
FUNCTION F_LogLA8 
VAR_INPUT
	eLogLevel		: E_LogLevel;
	sLogger			: T_MaxString;
	sMessage		: T_MaxString;
	aArg1			: ANY;
	aArg2			: ANY;
	aArg3			: ANY;
	aArg4			: ANY;
	aArg5			: ANY;
	aArg6			: ANY;
	aArg7			: ANY;
	aArg8			: ANY;
END_VAR
VAR 
	aEmptyArg		: BYTE;
END_VAR

F_LogA(
	eLogLevel,
	sLogger,
	sMessage,
	8,
	aArg1,
	aArg2,
	aArg3,
	aArg4,
	aArg5,
	aArg6,
	aArg7,
	aArg8,
	aEmptyArg,
	aEmptyArg,
	0
);

END_FUNCTION

// API/Simple/Any/F_LogA9
FUNCTION F_LogA9 
VAR_INPUT
	eLogLevel		: E_LogLevel;
	sMessage		: T_MaxString;
	aArg1			: ANY;
	aArg2			: ANY;
	aArg3			: ANY;
	aArg4			: ANY;
	aArg5			: ANY;
	aArg6			: ANY;
	aArg7			: ANY;
	aArg8			: ANY;
	aArg9			: ANY;
END_VAR

F_LogLA9(eLogLevel, Const.sGlobalLogger, sMessage, aArg1, aArg2, aArg3, aArg4, aArg5, aArg6, aArg7, aArg8, aArg9);

END_FUNCTION

// API/Simple/Any/F_LogLA9
FUNCTION F_LogLA9 
VAR_INPUT
	eLogLevel		: E_LogLevel;
	sLogger			: T_MaxString;
	sMessage		: T_MaxString;
	aArg1			: ANY;
	aArg2			: ANY;
	aArg3			: ANY;
	aArg4			: ANY;
	aArg5			: ANY;
	aArg6			: ANY;
	aArg7			: ANY;
	aArg8			: ANY;
	aArg9			: ANY;
END_VAR
VAR 
	aEmptyArg		: BYTE;
END_VAR

F_LogA(
	eLogLevel,
	sLogger,
	sMessage,
	9,
	aArg1,
	aArg2,
	aArg3,
	aArg4,
	aArg5,
	aArg6,
	aArg7,
	aArg8,
	aArg9,
	aEmptyArg,
	0
);

END_FUNCTION

// API/Simple/Any/F_LogLA10C
FUNCTION F_LogLA10C 
VAR_INPUT
	eLogLevel		: E_LogLevel;
	sLogger			: T_MaxString;
	sMessage		: T_MaxString;
	aArg1			: ANY;
	aArg2			: ANY;
	aArg3			: ANY;
	aArg4			: ANY;
	aArg5			: ANY;
	aArg6			: ANY;
	aArg7			: ANY;
	aArg8			: ANY;
	aArg9			: ANY;
	aArg10			: ANY;
	iContextBuilder	: I_ContextBuilder;
END_VAR

F_LogA(
	eLogLevel,
	sLogger,
	sMessage,
	10,
	aArg1,
	aArg2,
	aArg3,
	aArg4,
	aArg5,
	aArg6,
	aArg7,
	aArg8,
	aArg9,
	aArg10,
	iContextBuilder
);

END_FUNCTION

// API/Simple/Any/F_LogLA1C
FUNCTION F_LogLA1C 
VAR_INPUT
	eLogLevel		: E_LogLevel;
	sLogger			: T_MaxString;
	sMessage		: T_MaxString;
	aArg1			: ANY;
	iContextBuilder	: I_ContextBuilder;
END_VAR
VAR 
	aEmptyArg		: BYTE;
END_VAR

F_LogA(
	eLogLevel,
	sLogger,
	sMessage,
	1,
	aArg1,
	aEmptyArg,
	aEmptyArg,
	aEmptyArg,
	aEmptyArg,
	aEmptyArg,
	aEmptyArg,
	aEmptyArg,
	aEmptyArg,
	aEmptyArg,
	iContextBuilder
);

END_FUNCTION

// API/Simple/Any/F_LogLA2C
FUNCTION F_LogLA2C 
VAR_INPUT
	eLogLevel		: E_LogLevel;
	sLogger			: T_MaxString;
	sMessage		: T_MaxString;
	aArg1			: ANY;
	aArg2			: ANY;
	iContextBuilder	: I_ContextBuilder;
END_VAR
VAR 
	aEmptyArg		: BYTE;
END_VAR

F_LogA(
	eLogLevel,
	sLogger,
	sMessage,
	2,
	aArg1,
	aArg2,
	aEmptyArg,
	aEmptyArg,
	aEmptyArg,
	aEmptyArg,
	aEmptyArg,
	aEmptyArg,
	aEmptyArg,
	aEmptyArg,
	iContextBuilder
);

END_FUNCTION

// API/Simple/Any/F_LogLA3C
FUNCTION F_LogLA3C 
VAR_INPUT
	eLogLevel		: E_LogLevel;
	sLogger			: T_MaxString;
	sMessage		: T_MaxString;
	aArg1			: ANY;
	aArg2			: ANY;
	aArg3			: ANY;
	iContextBuilder	: I_ContextBuilder;
END_VAR
VAR 
	aEmptyArg		: BYTE;
END_VAR

F_LogA(
	eLogLevel,
	sLogger,
	sMessage,
	3,
	aArg1,
	aArg2,
	aArg3,
	aEmptyArg,
	aEmptyArg,
	aEmptyArg,
	aEmptyArg,
	aEmptyArg,
	aEmptyArg,
	aEmptyArg,
	iContextBuilder
);

END_FUNCTION

// API/Simple/Any/F_LogLA4C
FUNCTION F_LogLA4C 
VAR_INPUT
	eLogLevel		: E_LogLevel;
	sLogger			: T_MaxString;
	sMessage		: T_MaxString;
	aArg1			: ANY;
	aArg2			: ANY;
	aArg3			: ANY;
	aArg4			: ANY;
	iContextBuilder	: I_ContextBuilder;
END_VAR
VAR 
	aEmptyArg		: BYTE;
END_VAR

F_LogA(
	eLogLevel,
	sLogger,
	sMessage,
	4,
	aArg1,
	aArg2,
	aArg3,
	aArg4,
	aEmptyArg,
	aEmptyArg,
	aEmptyArg,
	aEmptyArg,
	aEmptyArg,
	aEmptyArg,
	iContextBuilder
);

END_FUNCTION

// API/Simple/Any/F_LogLA5C
FUNCTION F_LogLA5C 
VAR_INPUT
	eLogLevel		: E_LogLevel;
	sLogger			: T_MaxString;
	sMessage		: T_MaxString;
	aArg1			: ANY;
	aArg2			: ANY;
	aArg3			: ANY;
	aArg4			: ANY;
	aArg5			: ANY;
	iContextBuilder	: I_ContextBuilder;
END_VAR
VAR 
	aEmptyArg		: BYTE;
END_VAR

F_LogA(
	eLogLevel,
	sLogger,
	sMessage,
	5,
	aArg1,
	aArg2,
	aArg3,
	aArg4,
	aArg5,
	aEmptyArg,
	aEmptyArg,
	aEmptyArg,
	aEmptyArg,
	aEmptyArg,
	iContextBuilder
);

END_FUNCTION

// API/Simple/Any/F_LogLA6C
FUNCTION F_LogLA6C 
VAR_INPUT
	eLogLevel		: E_LogLevel;
	sLogger			: T_MaxString;
	sMessage		: T_MaxString;
	aArg1			: ANY;
	aArg2			: ANY;
	aArg3			: ANY;
	aArg4			: ANY;
	aArg5			: ANY;
	aArg6			: ANY;
	iContextBuilder	: I_ContextBuilder;
END_VAR
VAR 
	aEmptyArg		: BYTE;
END_VAR

F_LogA(
	eLogLevel,
	sLogger,
	sMessage,
	6,
	aArg1,
	aArg2,
	aArg3,
	aArg4,
	aArg5,
	aArg6,
	aEmptyArg,
	aEmptyArg,
	aEmptyArg,
	aEmptyArg,
	iContextBuilder
);

END_FUNCTION

// API/Simple/Any/F_LogLA7C
FUNCTION F_LogLA7C 
VAR_INPUT
	eLogLevel		: E_LogLevel;
	sLogger			: T_MaxString;
	sMessage		: T_MaxString;
	aArg1			: ANY;
	aArg2			: ANY;
	aArg3			: ANY;
	aArg4			: ANY;
	aArg5			: ANY;
	aArg6			: ANY;
	aArg7			: ANY;
	iContextBuilder	: I_ContextBuilder;
END_VAR
VAR 
	aEmptyArg		: BYTE;
END_VAR

F_LogA(
	eLogLevel,
	sLogger,
	sMessage,
	7,
	aArg1,
	aArg2,
	aArg3,
	aArg4,
	aArg5,
	aArg6,
	aArg7,
	aEmptyArg,
	aEmptyArg,
	aEmptyArg,
	iContextBuilder
);

END_FUNCTION

// API/Simple/Any/F_LogLA8C
FUNCTION F_LogLA8C 
VAR_INPUT
	eLogLevel		: E_LogLevel;
	sLogger			: T_MaxString;
	sMessage		: T_MaxString;
	aArg1			: ANY;
	aArg2			: ANY;
	aArg3			: ANY;
	aArg4			: ANY;
	aArg5			: ANY;
	aArg6			: ANY;
	aArg7			: ANY;
	aArg8			: ANY;
	iContextBuilder	: I_ContextBuilder;
END_VAR
VAR 
	aEmptyArg		: BYTE;
END_VAR

F_LogA(
	eLogLevel,
	sLogger,
	sMessage,
	8,
	aArg1,
	aArg2,
	aArg3,
	aArg4,
	aArg5,
	aArg6,
	aArg7,
	aArg8,
	aEmptyArg,
	aEmptyArg,
	iContextBuilder
);

END_FUNCTION

// API/Simple/Any/F_LogLA9C
FUNCTION F_LogLA9C 
VAR_INPUT
	eLogLevel		: E_LogLevel;
	sLogger			: T_MaxString;
	sMessage		: T_MaxString;
	aArg1			: ANY;
	aArg2			: ANY;
	aArg3			: ANY;
	aArg4			: ANY;
	aArg5			: ANY;
	aArg6			: ANY;
	aArg7			: ANY;
	aArg8			: ANY;
	aArg9			: ANY;
	iContextBuilder	: I_ContextBuilder;
END_VAR
VAR 
	aEmptyArg		: BYTE;
END_VAR

F_LogA(
	eLogLevel,
	sLogger,
	sMessage,
	9,
	aArg1,
	aArg2,
	aArg3,
	aArg4,
	aArg5,
	aArg6,
	aArg7,
	aArg8,
	aArg9,
	aEmptyArg,
	iContextBuilder
);

END_FUNCTION

// API/Simple/TArg/F_LogL1
FUNCTION F_LogL1 
VAR_INPUT
	eLogLevel		: E_LogLevel;
	sLogger			: T_MaxString;
	sMessage		: T_MaxString;
	stArg1			: T_Arg;

END_VAR

F_LogTArg(
	eLogLevel, 
	sLogger, 
	sMessage, 
	stArg1, 
	Tc2_Utilities.EMPTY_ARG_VALUE,  
	Tc2_Utilities.EMPTY_ARG_VALUE,  
	Tc2_Utilities.EMPTY_ARG_VALUE, 
	Tc2_Utilities.EMPTY_ARG_VALUE, 
	Tc2_Utilities.EMPTY_ARG_VALUE, 
	Tc2_Utilities.EMPTY_ARG_VALUE, 
	Tc2_Utilities.EMPTY_ARG_VALUE, 
	Tc2_Utilities.EMPTY_ARG_VALUE, 
	Tc2_Utilities.EMPTY_ARG_VALUE, 
	0
);

END_FUNCTION

// POUs/F_LogTArg
{attribute 'conditionalshow'}
FUNCTION INTERNAL F_LogTArg
VAR_INPUT
	eLogLevel		: E_LogLevel;
	sLogger			: Tc2_Utilities.T_MaxString;
	sMessage		: Tc2_Utilities.T_MaxString;
	stArg1			: Tc2_Utilities.T_Arg;
	stArg2			: Tc2_Utilities.T_Arg;
	stArg3			: Tc2_Utilities.T_Arg;
	stArg4			: Tc2_Utilities.T_Arg;
	stArg5			: Tc2_Utilities.T_Arg;
	stArg6			: Tc2_Utilities.T_Arg;
	stArg7			: Tc2_Utilities.T_Arg;
	stArg8			: Tc2_Utilities.T_Arg;
	stArg9			: Tc2_Utilities.T_Arg;
	stArg10			: Tc2_Utilities.T_Arg;
	iContextBuilder	: I_ContextBuilder;
END_VAR
VAR
	fbLogEntry			: FB_LogEntry();
	pBuffer				: PVOID;
	nBufferCount		: UINT;	
	iLogEntryAdder		: I_LogEntryAdder;
	nIdx				: UINT;
	refScopedContext	: REFERENCE TO ST_ScopedContextStack;
END_VAR

fbLogEntry.Start(
	pLogger			:= ADR(sLogger),
	pMessage		:= ADR(sMessage),
	eLogLevel		:= eLogLevel,
	nTimeStampPlc	:= 0,
	nTimeStampClock	:= 0
);

IF stArg1.eType <> Tc2_Utilities.E_ArgType.ARGTYPE_UNKNOWN AND stArg1.pData <> 0 THEN
	fbLogEntry.AddTArg(1, stArg1);
END_IF

IF stArg2.eType <> Tc2_Utilities.E_ArgType.ARGTYPE_UNKNOWN AND stArg2.pData <> 0 THEN
	fbLogEntry.AddTArg(2, stArg2);
END_IF

IF stArg3.eType <> Tc2_Utilities.E_ArgType.ARGTYPE_UNKNOWN AND stArg3.pData <> 0 THEN
	fbLogEntry.AddTArg(3, stArg3);
END_IF

IF stArg4.eType <> Tc2_Utilities.E_ArgType.ARGTYPE_UNKNOWN AND stArg4.pData <> 0 THEN
	fbLogEntry.AddTArg(4, stArg4);
END_IF

IF stArg5.eType <> Tc2_Utilities.E_ArgType.ARGTYPE_UNKNOWN AND stArg5.pData <> 0 THEN
	fbLogEntry.AddTArg(5, stArg5);
END_IF

IF stArg6.eType <> Tc2_Utilities.E_ArgType.ARGTYPE_UNKNOWN AND stArg6.pData <> 0 THEN
	fbLogEntry.AddTArg(6, stArg6);
END_IF

IF stArg7.eType <> Tc2_Utilities.E_ArgType.ARGTYPE_UNKNOWN AND stArg7.pData <> 0 THEN
	fbLogEntry.AddTArg(7, stArg7);
END_IF

IF stArg8.eType <> Tc2_Utilities.E_ArgType.ARGTYPE_UNKNOWN AND stArg8.pData <> 0 THEN
	fbLogEntry.AddTArg(8, stArg8);
END_IF

IF stArg9.eType <> Tc2_Utilities.E_ArgType.ARGTYPE_UNKNOWN AND stArg9.pData <> 0 THEN
	fbLogEntry.AddTArg(9, stArg9);
END_IF

IF stArg10.eType <> Tc2_Utilities.E_ArgType.ARGTYPE_UNKNOWN AND stArg10.pData <> 0 THEN
	fbLogEntry.AddTArg(10, stArg10);
END_IF

IF __QUERYINTERFACE(PRG_TaskLog.TaskLogger.TaskContext, iLogEntryAdder) THEN
	iLogEntryAdder.AddToLogEntry(E_Scope.eTask, fbLogEntry);
END_IF

refScopedContext REF= PRG_ScopedContextStack.TaskContextStack;
FOR nIdx := 0 TO refScopedContext.nScopeContextCount - 1 DO
	IF __QUERYINTERFACE(refScopedContext.aScopedContext[nIdx], iLogEntryAdder) THEN
		iLogEntryAdder.AddToLogEntry(E_Scope.eScoped, fbLogEntry);
	END_IF
END_FOR

IF iContextBuilder <> 0 AND __QUERYINTERFACE(iContextBuilder, iLogEntryAdder) THEN
	iLogEntryAdder.AddToLogEntry(E_Scope.eLogger, fbLogEntry);
END_IF

fbLogEntry.End();

END_FUNCTION

// API/Simple/TArg/F_LogL10
FUNCTION F_LogL10 
VAR_INPUT
	eLogLevel		: E_LogLevel;
	sLogger			: T_MaxString;
	sMessage		: T_MaxString;
	stArg1			: T_Arg;
	stArg2			: T_Arg;
	stArg3			: T_Arg;
	stArg4			: T_Arg;
	stArg5			: T_Arg;
	stArg6			: T_Arg;
	stArg7			: T_Arg;
	stArg8			: T_Arg;
	stArg9			: T_Arg;
	stArg10			: T_Arg;
END_VAR

F_LogTArg(
	eLogLevel, 
	sLogger, 
	sMessage, 
	stArg1, 
	stArg2, 
	stArg3, 
	stArg4, 
	stArg5, 
	stArg6, 
	stArg7, 
	stArg8, 
	stArg9, 
	stArg10, 
	0
);

END_FUNCTION

// API/Simple/TArg/F_LogL2
FUNCTION F_LogL2 
VAR_INPUT
	eLogLevel		: E_LogLevel;
	sLogger			: T_MaxString;
	sMessage		: T_MaxString;
	stArg1			: T_Arg;
	stArg2			: T_Arg;
END_VAR

F_LogTArg(
	eLogLevel, 
	sLogger, 
	sMessage, 
	stArg1, 
	stArg2, 
	Tc2_Utilities.EMPTY_ARG_VALUE, 
	Tc2_Utilities.EMPTY_ARG_VALUE, 
	Tc2_Utilities.EMPTY_ARG_VALUE, 
	Tc2_Utilities.EMPTY_ARG_VALUE, 
	Tc2_Utilities.EMPTY_ARG_VALUE, 
	Tc2_Utilities.EMPTY_ARG_VALUE, 
	Tc2_Utilities.EMPTY_ARG_VALUE, 
	Tc2_Utilities.EMPTY_ARG_VALUE, 
	0
);

END_FUNCTION

// API/Simple/TArg/F_LogL3
FUNCTION F_LogL3 
VAR_INPUT
	eLogLevel		: E_LogLevel;
	sLogger			: T_MaxString;
	sMessage		: T_MaxString;
	stArg1			: T_Arg;
	stArg2			: T_Arg;
	stArg3			: T_Arg;
END_VAR

F_LogTArg(
	eLogLevel, 
	sLogger, 
	sMessage, 
	stArg1, 
	stArg2, 
	stArg3, 
	Tc2_Utilities.EMPTY_ARG_VALUE, 
	Tc2_Utilities.EMPTY_ARG_VALUE, 
	Tc2_Utilities.EMPTY_ARG_VALUE, 
	Tc2_Utilities.EMPTY_ARG_VALUE, 
	Tc2_Utilities.EMPTY_ARG_VALUE, 
	Tc2_Utilities.EMPTY_ARG_VALUE, 
	Tc2_Utilities.EMPTY_ARG_VALUE, 
	0
);

END_FUNCTION

// API/Simple/TArg/F_LogL4
FUNCTION F_LogL4 
VAR_INPUT
	eLogLevel		: E_LogLevel;
	sLogger			: T_MaxString;
	sMessage		: T_MaxString;
	stArg1			: T_Arg;
	stArg2			: T_Arg;
	stArg3			: T_Arg;
	stArg4			: T_Arg;
END_VAR

F_LogTArg(
	eLogLevel, 
	sLogger, 
	sMessage, 
	stArg1, 
	stArg2, 
	stArg3, 
	stArg4, 
	Tc2_Utilities.EMPTY_ARG_VALUE, 
	Tc2_Utilities.EMPTY_ARG_VALUE, 
	Tc2_Utilities.EMPTY_ARG_VALUE, 
	Tc2_Utilities.EMPTY_ARG_VALUE, 
	Tc2_Utilities.EMPTY_ARG_VALUE, 
	Tc2_Utilities.EMPTY_ARG_VALUE, 
	0
);

END_FUNCTION

// API/Simple/TArg/F_LogL5
FUNCTION F_LogL5 
VAR_INPUT
	eLogLevel		: E_LogLevel;
	sLogger			: T_MaxString;
	sMessage		: T_MaxString;
	stArg1			: T_Arg;
	stArg2			: T_Arg;
	stArg3			: T_Arg;
	stArg4			: T_Arg;
	stArg5			: T_Arg;
END_VAR

F_LogTArg(
	eLogLevel, 
	sLogger, 
	sMessage, 
	stArg1, 
	stArg2, 
	stArg3, 
	stArg4, 
	stArg5, 
	Tc2_Utilities.EMPTY_ARG_VALUE, 
	Tc2_Utilities.EMPTY_ARG_VALUE, 
	Tc2_Utilities.EMPTY_ARG_VALUE, 
	Tc2_Utilities.EMPTY_ARG_VALUE, 
	Tc2_Utilities.EMPTY_ARG_VALUE, 
	0
);

END_FUNCTION

// API/Simple/TArg/F_LogL6
FUNCTION F_LogL6 
VAR_INPUT
	eLogLevel		: E_LogLevel;
	sLogger			: T_MaxString;
	sMessage		: T_MaxString;
	stArg1			: T_Arg;
	stArg2			: T_Arg;
	stArg3			: T_Arg;
	stArg4			: T_Arg;
	stArg5			: T_Arg;
	stArg6			: T_Arg;
END_VAR

F_LogTArg(
	eLogLevel, 
	sLogger, 
	sMessage, 
	stArg1, 
	stArg2, 
	stArg3, 
	stArg4, 
	stArg5, 
	stArg6, 
	Tc2_Utilities.EMPTY_ARG_VALUE, 
	Tc2_Utilities.EMPTY_ARG_VALUE, 
	Tc2_Utilities.EMPTY_ARG_VALUE, 
	Tc2_Utilities.EMPTY_ARG_VALUE, 
	0
);

END_FUNCTION

// API/Simple/TArg/F_LogL7
FUNCTION F_LogL7 
VAR_INPUT
	eLogLevel		: E_LogLevel;
	sLogger			: T_MaxString;
	sMessage		: T_MaxString;
	stArg1			: T_Arg;
	stArg2			: T_Arg;
	stArg3			: T_Arg;
	stArg4			: T_Arg;
	stArg5			: T_Arg;
	stArg6			: T_Arg;
	stArg7			: T_Arg;
END_VAR

F_LogTArg(
	eLogLevel, 
	sLogger, 
	sMessage, 
	stArg1, 
	stArg2, 
	stArg3, 
	stArg4, 
	stArg5, 
	stArg6, 
	stArg7, 
	Tc2_Utilities.EMPTY_ARG_VALUE, 
	Tc2_Utilities.EMPTY_ARG_VALUE, 
	Tc2_Utilities.EMPTY_ARG_VALUE, 
	0
);

END_FUNCTION

// API/Simple/TArg/F_LogL8
FUNCTION F_LogL8 
VAR_INPUT
	eLogLevel		: E_LogLevel;
	sLogger			: T_MaxString;
	sMessage		: T_MaxString;
	stArg1			: T_Arg;
	stArg2			: T_Arg;
	stArg3			: T_Arg;
	stArg4			: T_Arg;
	stArg5			: T_Arg;
	stArg6			: T_Arg;
	stArg7			: T_Arg;
	stArg8			: T_Arg;
END_VAR

F_LogTArg(
	eLogLevel, 
	sLogger, 
	sMessage, 
	stArg1, 
	stArg2, 
	stArg3, 
	stArg4, 
	stArg5, 
	stArg6, 
	stArg7, 
	stArg8, 
	Tc2_Utilities.EMPTY_ARG_VALUE, 
	Tc2_Utilities.EMPTY_ARG_VALUE, 
	0
);

END_FUNCTION

// API/Simple/TArg/F_LogL9
FUNCTION F_LogL9 
VAR_INPUT
	eLogLevel		: E_LogLevel;
	sLogger			: T_MaxString;
	sMessage		: T_MaxString;
	stArg1			: T_Arg;
	stArg2			: T_Arg;
	stArg3			: T_Arg;
	stArg4			: T_Arg;
	stArg5			: T_Arg;
	stArg6			: T_Arg;
	stArg7			: T_Arg;
	stArg8			: T_Arg;
	stArg9			: T_Arg;
END_VAR

F_LogTArg(
	eLogLevel, 
	sLogger, 
	sMessage, 
	stArg1, 
	stArg2, 
	stArg3, 
	stArg4, 
	stArg5, 
	stArg6, 
	stArg7, 
	stArg8, 
	stArg9, 
	Tc2_Utilities.EMPTY_ARG_VALUE, 
	0
);

END_FUNCTION

// API/Simple/F_Log
(*
:Description: Writes the given message at the specific level. 

This function implicit uses the global logger ``Const.sGlobalLogger`` with
the value ``'_GLOBAL_'``.

**Example**

.. code:: 

    F_Log(E_LogLevel.eWarn, 'Something important happened.');
	
*)
FUNCTION F_Log
VAR_INPUT
	eLogLevel		: E_LogLevel;		(* The level of this log. *)
	sMessage		: T_MaxString;		(* The message to log. *)
END_VAR
VAR 
	aEmptyArg		: BYTE;
END_VAR

F_LogL(eLogLevel, Const.sGlobalLogger, sMessage);

END_FUNCTION

// API/Simple/F_LogL
(*
:Description: Writes the given message at the specific level and logger name. 

**Logger**

The logger is used to give the message a scope. Although not enforced, it is
recommended to use a hierarchical structure which reflects the code. For example
if the method ``CheckTemp`` of a program block ``PRG_Alarms`` is writing a log message,
the logger name could be ``'PRG_Alarms.CheckTemp'``.

**Example**

.. code:: 

    F_LogL(E_LogLevel.eWarn, 'PRG_Alarms' ,'Something important happened.');
	
*)
FUNCTION F_LogL : BOOL
VAR_INPUT
	eLogLevel		: E_LogLevel;		(* The level of this log. *)
	sLogger			: T_MaxString;      (* The name of the logger. *)
	sMessage		: T_MaxString;		(* The message to log. *)
END_VAR
VAR 
	aEmptyArg		: BYTE;
END_VAR

F_LogA(eLogLevel, sLogger, sMessage, 0, aEmptyArg, aEmptyArg, aEmptyArg, aEmptyArg, aEmptyArg, aEmptyArg, aEmptyArg, aEmptyArg, aEmptyArg, aEmptyArg, 0);

END_FUNCTION

// API/Simple/F_LogBuilder
FUNCTION F_LogBuilder : I_LogBuilder
VAR_INPUT
	eLogLevel		: E_LogLevel;
	sMessages		: T_MaxString;
END_VAR

END_FUNCTION

// API/Simple/I_LogBuilder
INTERFACE I_LogBuilder

METHOD CreateLog
END_METHOD

METHOD WithContextInt : I_LogBuilder
VAR_INPUT
	sName		: T_MaxString;
	nValue		: INT;
END_VAR
END_METHOD

METHOD WithIntArg : I_LogBuilder
VAR_INPUT
	nValue		: INT;
END_VAR
END_METHOD

METHOD WithLogger : I_LogBuilder
VAR_INPUT
	sLogger		: T_MaxString;
END_VAR
END_METHOD

METHOD WithStringArg : I_LogBuilder
VAR_INPUT
	sValue		: T_MaxString;
END_VAR
END_METHOD

END_INTERFACE

// API/Simple/F_LogC
(*
:Description: Writes the given message at the specific level, on the Global logger name and with
	the given context properties. 

**Logger**

The logger is used to give the message a scope. Although not enforced, it is
recommended to use a hierarchical structure which reflects the code. For example
if the method ``CheckTemp`` of a program block ``PRG_Alarms`` is writing a log message,
the logger name could be ``'PRG_Alarms.CheckTemp'``.

**Example**

.. code:: 

    F_LogC(E_LogLevel.eWarn, 'Something important happened.', F_LogContext().AddInt('serial', 1234));
	
*)
FUNCTION F_LogC : BOOL
VAR_INPUT
	eLogLevel		: E_LogLevel;		(* The level of this log. *)
	sMessage		: T_MaxString;		(* The message to log. *)
	iContextBuilder	: I_ContextBuilder;	(* A context builder (or 0) *)
END_VAR
VAR 
	aEmptyArg		: BYTE;
END_VAR

F_LogA(eLogLevel, Const.sGlobalLogger, sMessage, 0, aEmptyArg, aEmptyArg, aEmptyArg, aEmptyArg, aEmptyArg, aEmptyArg, aEmptyArg, aEmptyArg, aEmptyArg, aEmptyArg, iContextBuilder);

END_FUNCTION

// API/Simple/F_LogLC
(*
:Description: Writes the given message at the specific level, logger name and with
	the given context properties. 

**Logger**

The logger is used to give the message a scope. Although not enforced, it is
recommended to use a hierarchical structure which reflects the code. For example
if the method ``CheckTemp`` of a program block ``PRG_Alarms`` is writing a log message,
the logger name could be ``'PRG_Alarms.CheckTemp'``.

**Example**

.. code:: 

    F_LogLC(E_LogLevel.eWarn, 'PRG_Alarms' ,'Something important happened.', F_LogContext().AddInt('serial', 1234));
	
*)
FUNCTION F_LogLC : BOOL
VAR_INPUT
	eLogLevel		: E_LogLevel;		(* The level of this log. *)
	sLogger			: T_MaxString;      (* The name of the logger. *)
	sMessage		: T_MaxString;		(* The message to log. *)
	iContextBuilder	: I_ContextBuilder;	(* A context builder (or 0) *)
END_VAR
VAR 
	aEmptyArg		: BYTE;
END_VAR

F_LogA(eLogLevel, sLogger, sMessage, 0, aEmptyArg, aEmptyArg, aEmptyArg, aEmptyArg, aEmptyArg, aEmptyArg, aEmptyArg, aEmptyArg, aEmptyArg, aEmptyArg, iContextBuilder);

END_FUNCTION

// POUs/Utils/F_DINT_TO_UINT_MAX
FUNCTION INTERNAL F_DINT_TO_UINT_MAX : UINT
VAR_INPUT
	nValue			: DINT;
	nMaxValue		: UINT;
END_VAR

IF nValue < 0 THEN
	F_DINT_TO_UINT_MAX := 0;
ELSIF nValue > nMaxValue THEN
	F_DINT_TO_UINT_MAX := nMaxValue;
ELSE
	F_DINT_TO_UINT_MAX := DINT_TO_UINT(nValue);
END_IF

END_FUNCTION

// Test/FB_ContextBuilder_Test
FUNCTION_BLOCK INTERNAL FB_ContextBuilder_Test EXTENDS TcUnit.FB_TestSuite

AddInt_ShouldAddInt();
AddInt_WithSameName_ShouldReplace();
RemoveInt_ShouldRemove();

AddString_ShouldAddString();
AddString_WithSameName_ShouldReAdd();
AddString_WithSameName_ShouldReplace();
RemoveString_ShouldRemove();

METHOD AddInt_ShouldAddInt
VAR
	fbContextBuilder		: FB_ContextBuilder;
END_VAR
TcUnit.TEST('AddInt_ShouldAddInt');

fbContextBuilder.AddInt('foo', 42);

// 1 + 'foo' + 2 + 2
AssertEquals_UINT(8, fbContextBuilder._BufferCount, 'Buffer size');
AssertEquals_UINT(1, fbContextBuilder._ContextCount, 'Context count');
AssertEquals_UINT(0, fbContextBuilder._GetContextOffset(0), 'Context[0]');
AssertEquals_STRING('foo', fbContextBuilder._ReadName(0), 'Name');
AssertEquals_INT(Tc2_Utilities.E_ArgType.ARGTYPE_INT, fbContextBuilder._ReadType(0), 'Type');

TcUnit.TEST_FINISHED();
END_METHOD

METHOD AddInt_WithSameName_ShouldReplace
VAR
	fbContextBuilder		: FB_ContextBuilder;

END_VAR
TcUnit.TEST('AddInt_WithSameName_ShouldReplace');

// first add some
fbContextBuilder.AddInt('before', 0);	// size: 11
fbContextBuilder.AddWord('foo', 42);	// size: 8
fbContextBuilder.AddInt('after', 0);	// size: 10

// then replace
fbContextBuilder.AddInt('foo', 0);

AssertEquals_UINT(29, fbContextBuilder._BufferCount, 'Buffer size');
AssertEquals_UINT(3, fbContextBuilder._ContextCount, 'Context count');
AssertEquals_UINT(0, fbContextBuilder._GetContextOffset(0), 'Context[0]');
AssertEquals_UINT(11, fbContextBuilder._GetContextOffset(1), 'Context[1]');
AssertEquals_UINT(19, fbContextBuilder._GetContextOffset(2), 'Context[2]');
AssertEquals_STRING('before', fbContextBuilder._ReadName(0), 'Name[0]');
AssertEquals_STRING('foo', fbContextBuilder._ReadName(1), 'Name[1]');
AssertEquals_STRING('after', fbContextBuilder._ReadName(2), 'Name[2]');
AssertEquals_INT(Tc2_Utilities.E_ArgType.ARGTYPE_INT, fbContextBuilder._ReadType(1), 'Type');

TcUnit.TEST_FINISHED();
END_METHOD

METHOD AddString_ShouldAddString
VAR
	fbContextBuilder		: FB_ContextBuilder;
END_VAR
TcUnit.TEST('AddString_ShouldAddString');

fbContextBuilder.AddString('foo', 'bar');	// size: 10

AssertEquals_UINT(10, fbContextBuilder._BufferCount, 'Buffer size');
AssertEquals_UINT(1, fbContextBuilder._ContextCount, 'Context count');
AssertEquals_UINT(0, fbContextBuilder._GetContextOffset(0), 'Context[0]');
AssertEquals_STRING('foo', fbContextBuilder._ReadName(0), 'Name');
AssertEquals_INT(Tc2_Utilities.E_ArgType.ARGTYPE_STRING, fbContextBuilder._ReadType(0), 'Type');

TcUnit.TEST_FINISHED();
END_METHOD

METHOD AddString_WithSameName_ShouldReAdd
VAR
	fbContextBuilder		: FB_ContextBuilder;
END_VAR
TcUnit.TEST('AddString_WithSameName_ShouldReAdd');

fbContextBuilder.AddString('before', 'aaa');	// Size: 13
fbContextBuilder.AddString('foo', 'bar');		// Size: 10
fbContextBuilder.AddString('after', 'zzz');		// Size: 12

fbContextBuilder.AddString('foo', 'bazbar');	// Size: 13

AssertEquals_UINT(38, fbContextBuilder._BufferCount, 'Buffer size');
AssertEquals_UINT(3, fbContextBuilder._ContextCount, 'Context count');
AssertEquals_UINT(0, fbContextBuilder._GetContextOffset(0), 'Context[0]');
AssertEquals_UINT(13, fbContextBuilder._GetContextOffset(1), 'Context[1]');
AssertEquals_UINT(25, fbContextBuilder._GetContextOffset(2), 'Context[2]');
AssertEquals_STRING('before', fbContextBuilder._ReadName(0), 'Name[0]');
AssertEquals_STRING('after', fbContextBuilder._ReadName(1), 'Name[1]');
AssertEquals_STRING('foo', fbContextBuilder._ReadName(2), 'Name[2]');
AssertEquals_INT(Tc2_Utilities.E_ArgType.ARGTYPE_STRING, fbContextBuilder._ReadType(2), 'Type');

TcUnit.TEST_FINISHED();
END_METHOD

METHOD AddString_WithSameName_ShouldReplace
VAR
	fbContextBuilder		: FB_ContextBuilder;
END_VAR
TcUnit.TEST('AddString_WithSameName_ShouldReplace');

fbContextBuilder.AddString('before', 'aaa');	// Size: 13
fbContextBuilder.AddString('foo', 'bar');		// Size: 10
fbContextBuilder.AddString('after', 'zzz');		// Size: 12

fbContextBuilder.AddString('foo', 'baz');

AssertEquals_UINT(35, fbContextBuilder._BufferCount, 'Buffer size');
AssertEquals_UINT(3, fbContextBuilder._ContextCount, 'Context count');
AssertEquals_UINT(0, fbContextBuilder._GetContextOffset(0), 'Context[0]');
AssertEquals_UINT(13, fbContextBuilder._GetContextOffset(1), 'Context[1]');
AssertEquals_UINT(23, fbContextBuilder._GetContextOffset(2), 'Context[2]');
AssertEquals_STRING('before', fbContextBuilder._ReadName(0), 'Name[0]');
AssertEquals_STRING('foo', fbContextBuilder._ReadName(1), 'Name[1]');
AssertEquals_STRING('after', fbContextBuilder._ReadName(2), 'Name[2]');
AssertEquals_INT(Tc2_Utilities.E_ArgType.ARGTYPE_STRING, fbContextBuilder._ReadType(2), 'Type');

TcUnit.TEST_FINISHED();
END_METHOD

METHOD RemoveInt_ShouldRemove
VAR
	fbContextBuilder		: FB_ContextBuilder;

END_VAR
TcUnit.TEST('RemoveInt_ShouldRemove');

// first add some
fbContextBuilder.AddInt('before', 0);	// size: 11
fbContextBuilder.AddWord('foo', 42);	// size: 8
fbContextBuilder.AddInt('after', 0);	// size: 10

// then remove
fbContextBuilder.Remove('foo');

AssertEquals_UINT(21, fbContextBuilder._BufferCount, 'Buffer size');
AssertEquals_UINT(2, fbContextBuilder._ContextCount, 'Context count');
AssertEquals_UINT(0, fbContextBuilder._GetContextOffset(0), 'Context[0]');
AssertEquals_UINT(11, fbContextBuilder._GetContextOffset(1), 'Context[1]');
AssertEquals_STRING('before', fbContextBuilder._ReadName(0), 'Name[0]');
AssertEquals_STRING('after', fbContextBuilder._ReadName(1), 'Name[1]');

TcUnit.TEST_FINISHED();
END_METHOD

METHOD RemoveString_ShouldRemove
VAR
	fbContextBuilder		: FB_ContextBuilder;
END_VAR
TcUnit.TEST('RemoveString_ShouldRemove');

fbContextBuilder.AddString('before', 'aaa');	// Size: 13
fbContextBuilder.AddString('foo', 'bar');		// Size: 10
fbContextBuilder.AddString('after', 'zzz');		// Size: 12

fbContextBuilder.Remove('foo');

AssertEquals_UINT(25, fbContextBuilder._BufferCount, 'Buffer size');
AssertEquals_UINT(2, fbContextBuilder._ContextCount, 'Context count');
AssertEquals_UINT(0, fbContextBuilder._GetContextOffset(0), 'Context[0]');
AssertEquals_UINT(13, fbContextBuilder._GetContextOffset(1), 'Context[1]');
AssertEquals_STRING('before', fbContextBuilder._ReadName(0), 'Name[0]');
AssertEquals_STRING('after', fbContextBuilder._ReadName(1), 'Name[1]');

TcUnit.TEST_FINISHED();
END_METHOD

END_FUNCTION_BLOCK

// Test/PRG_Test
PROGRAM INTERNAL PRG_Test
VAR
	fbContextBuilder_Test	: FB_ContextBuilder_Test;
	
	fbLog			: FB_LoggerLAC(Const.sLoggerFromInstance);
	
	fbScope			: FB_ScopedContext;
	bLog			: BOOL;
	bArg1			: BOOL;
	nArg2			: INT;
	sArg3			: STRING;
	
	
END_VAR

TcUnit.RUN();

IF _TaskInfo[GETCURTASKINDEXEX()].FirstCycle THEN
	// For Remote Log4TC Server change the AMS net ID and configure a route
	PRG_TaskLog.Init('127.0.0.1.1.1');
	F_Log(E_LogLevel.eInfo, 'SPS Task gestartet.');
END_IF

fbLog.LoggerContext.AddInt('logger', 42);

IF bLog THEN
	bLog := FALSE;
	F_Log(E_LogLevel.eDebug, 'Foobar'); 
	F_LogA3(E_LogLevel.eInfo, '{0}, {1}, {2}', bArg1, nArg2, sArg3);

	fbLog(
		eLogLevel 		:= E_LogLevel.eInfo,
		sMessage 		:= 'barbaz {bLog}',
		aArg1 			:= bLog,
		iContextBuilder := F_LogContext().AddString('inmessage', 'foo')
	);
END_IF

PRG_TaskLog.Call();

END_PROGRAM

// ApiTest
PROGRAM INTERNAL ApiTest
VAR
	nInt			: INT;
	sStr			: STRING;
	fFloat			: REAL;
END_VAR

// Einfaches Logging
F_LogLC(
	E_LogLevel.eInfo,
	'ApiTest',
	'Log message',
	0
);

F_LogL3(
	E_LogLevel.eInfo,
	Const.sGlobalLogger, 
	'Log Message Arg={structuredArg} Arg={1} Arg=%s', 
	F_StringEx('Arg 1'),
	F_StringEx('Arg 2'),
	F_StringEx('Arg 3')
);

F_LogA3(
	E_LogLevel.eError,
	'Log Message Arg={structuredArg} Arg={1} Arg=%s',
	nInt,
	sStr,
	fFloat
);

// Einfaches Logging mit expliziten Logger
F_LogL3(
	E_LogLevel.eInfo, 
	'mbc4Log.Test',
	'Log Message Arg={structuredArg} Arg={1} Arg=%s', 
	F_StringEx('Arg 1'),
	F_StringEx('Arg 2'),
	F_StringEx('Arg 3')
);

// Einfaches Logging mit Builder
F_LogBuilder(E_LogLevel.eError, 'Log Message Arg={structuredArg} Arg={1} Arg=%s')
	.WithIntArg(42).WithStringArg('Arg 2').WithStringArg('Arg 3')
	.WithLogger('mbc4Log.Test')
	.WithContextInt('id', 42)
	.CreateLog();

END_PROGRAM
